// TwinCAT 3 PLC project MasterController
// ProgramVersion: 3.1.4024.0
// libraries:
//   Tc2_EtherCAT, * (Beckhoff Automation GmbH)
//   Tc2_Math, * (Beckhoff Automation GmbH)
//   Tc2_Standard, * (Beckhoff Automation GmbH)
//   Tc2_System, * (Beckhoff Automation GmbH)
//   Tc2_Utilities, * (Beckhoff Automation GmbH)
//   Tc3_Module, * (Beckhoff Automation GmbH)
// project tree:
//   AgiMaths/Frames/ DHTrans.TcPOU (not stored), invFrame.TcPOU, rotX.TcPOU, rotY.TcPOU, rotZ.TcPOU, transform.TcPOU
//   AgiMaths/MatrixLib/ angAxis2Rot.TcPOU, cross.TcPOU (not stored), Det5.TcPOU, Det6.TcPOU, Det7.TcPOU (not stored), invMat6.TcPOU, invMat6Old.TcPOU (not stored), invMat3.TcPOU, invMat7.TcPOU, Mat3T.TcPOU (not stored), matAdd.TcPOU, matMultiNum.TcPOU, matMultiply.TcPOU, matMultiVec.TcPOU, matSelfAdd.TcPOU, matSelfSub.TcPOU, matSub.TcPOU, matTranspose.TcPOU, rot2AngAxis.TcPOU, norm.TcPOU, normalize.TcPOU, vecAdd.TcPOU, vecDot.TcPOU, vecMultiNum.TcPOU, vecSelfAdd.TcPOU, vecSelfMultiNum.TcPOU, vecSelfSub.TcPOU, vecSub.TcPOU
//   AgiMaths/ sign.TcPOU (not stored), addVec7.TcPOU (not stored), atan2.TcPOU, cot.TcPOU (not stored)
//   DUTs/Enum/ E_InstruEnergyCtrlWord.TcDUT, E_InstrumentEnergyType.TcDUT, E_InstrumentType.TcDUT, E_MasterArmState.TcDUT, E_MatchedSlaveArmIdx.TcDUT (not stored), E_SlaveArmState.TcDUT, E_DriverCtrlWord.TcDUT (not stored), E_DriverOPMode.TcDUT, E_DriverStatusWord.TcDUT (not stored)
//   DUTs/Structure/MasterSlaveCommunication/ ST_MasterStatus.TcDUT, ST_SlaveStatus.TcDUT
//   DUTs/Structure/ ST_EtherCATState.TcDUT, ST_InstruStatus.TcDUT, ST_MatchedMasterArmIdx.TcDUT, ST_ArmCtrlCmds.TcDUT (not stored), ST_MasterInputDataPool.TcDUT, ST_Frame.TcDUT (not stored)
//   DUTs/Structure/TasksCommunication/ ST_CartUIData.TcDUT, ST_MasterDynaData.TcDUT, ST_MasterUIData.TcDUT, ST_CartStatus.TcDUT, ST_MasterJointData.TcDUT, ST_MotorInputs.TcDUT (not stored), ST_MotorOutputs.TcDUT, ST_SlaveJointData.TcDUT, ST_SafetyData.TcDUT, ST_CartJointData.TcDUT
//   DUTs/Structure/UICommunication/ ST_arm_distribution.TcDUT, ST_ergonCtrlEnable.TcDUT, ST_ergonomicCtrlData.TcDUT, ST_instrument_info.TcDUT, ST_scope_info.TcDUT
//   DUTs/Type/ Vec7b.TcDUT, Mat34.TcDUT, Mat37.TcDUT, Mat43.TcDUT, Mat4d.TcDUT, Mat5d.TcDUT, Mat67.TcDUT (not stored), Mat6d.TcDUT (not stored), Mat76.TcDUT (not stored), Mat7d.TcDUT (not stored), Vec4d.TcDUT, Vec4i.TcDUT, Vec6i.TcDUT, Vec4b.TcDUT, Vec7di.TcDUT, Vec8d.TcDUT, Mat3d.TcDUT (not stored), Vec3d.TcDUT (not stored), Vec6d.TcDUT (not stored), Vec7d.TcDUT, Vec7i.TcDUT
//   FBs_Auxiliary/ FB_GripAngleCalc.TcPOU, FB_HandClutchCheck.TcPOU, FB_IOCheck.TcPOU, FB_RiseEdgeCheck.TcPOU, FB_IOToggleCheck.TcPOU, FB_MSCtrlTriggerCheck.TcPOU, FB_slaveConnectionCheck.TcPOU, FB_TON.TcPOU
//   FBs_BasicControllers/ FB_boundaryForceFeedback.TcPOU, FB_PID.TcPOU (not stored), FB_RedunJntControl.TcPOU
//   FBs_Observer/ FB_JntObserver.TcPOU
//   FBs_RobotDynamics/ FB_MasterDynamic.TcPOU, FB_MasterFriciton.TcPOU, FB_MasterGravity.TcPOU
//   FBs_Robots/ FB_ArmJoint.TcPOU, FB_CartJoint.TcPOU, FB_JointBase.TcPOU, FB_MasterCart.TcPOU, FB_MasterArm.TcPOU, FB_MasterRobot.TcPOU
//   FBs_StateControllers/ FB_EndoscopeController.TcPOU, FB_StateCtrlClutch.TcPOU, FB_StateCtrlEndoscope.TcPOU, FB_StateCtrlCart.TcPOU, FB_StateCtrlDisable.TcPOU, FB_StateCtrlGraCali.TcPOU, FB_StateCtrlMatching.TcPOU, FB_StateCtrlHome.TcPOU, FB_StateCtrlError.TcPOU, FB_StateCtrlPerformance.TcPOU, FB_StateCtrlReady.TcPOU, FB_StateCtrlMasterSlave.TcPOU, FB_StateCtrlTest.TcPOU, FB_StateCtrlInit.TcPOU, FB_StateCtrlStandBy.TcPOU, FB_MasterArmCtrlBase.TcPOU, I_MasterArmCtrl.TcIO
//   FBs_TrajectoryPlanning/ FB_BasicDoubleS.TcPOU, FB_trajBase.TcPOU, FB_TrajMoveJ.TcPOU, linear_trajectory_with_quintic_polynomial_blends.TcPOU (not stored), quintic_spline_curve.TcPOU (not stored), Quintic_spline_curve_factor.TcPOU (not stored), TrapezoIDal_velocity_trajectory.TcPOU (not stored)
//   FBs_TrajectoryPlanning/OTG/ FB_secOrdTrajFilter.TcPOU, FB_thirdOrdTrajFilter.TcPOU (not stored)
//   FBs_Filters/ FB_LowPassFilter.TcPOU
//   GVLs/Arms/ GVL_ArmDynamics.TcGVL, GVL_ArmJointCaliData.TcGVL, GVL_ArmKinematic.TcGVL, GVL_ControlParameters.TcGVL, GVL_ArmJointParameters.TcGVL
//   GVLs/Cart/ GVL_CartJointCaliData.TcGVL, GVL_CartJointParameters.TcGVL
//   GVLs/Configs/Robot3/ GVL_ArmDynamics_3.TcGVL, GVL_ArmJointCaliData_3.TcGVL, GVL_CartJointCaliData_3.TcGVL
//   GVLs/Configs/Robot4/ GVL_ArmDynamics_4.TcGVL, GVL_ArmJointCaliData_4.TcGVL, GVL_CartJointCaliData_4_1.TcGVL
//   GVLs/Configs/Robot5/ GVL_ArmDynamics_5.TcGVL, GVL_ArmJointCaliData_5.TcGVL, GVL_CartJointCaliData_5.TcGVL
//   GVLs/Configs/Robot6/ GVL_ArmDynamics_6.TcGVL, GVL_ArmJointCaliData_6.TcGVL, GVL_CartJointCaliData_6.TcGVL
//   GVLs/ GVL_interactUI.TcGVL, GVL_MathDefine.TcGVL, GVL_SafetyParameters.TcGVL, GVL_SystemParameters.TcGVL
//   Mains/ CartControl.TcPOU, SafetyCheck.TcPOU, MasterArmControl.TcPOU, RobotDynamics.TcPOU
//   SafetyCheck/ ASSERT.TcPOU, Fb_dataRecord.TcPOU, FB_EtherCATCheck.TcPOU, Fb_SafetyCheck.TcPOU, FB_Writer.TcPOU
//   SafetyCheck/safetyCheckDUT/ checkDelay.TcDUT, checkDelayTime.TcDUT, checkInputVariable.TcDUT, checkPermit.TcDUT, ST_Buffer.TcDUT, T_Buffer.TcDUT
//   Sandbox/ FB_CartCheck.TcPOU, FB_MasterArmCheck.TcPOU, FB_RedunJntControl_bak2.TcPOU, FB_RedunJntControl_bak.TcPOU
//   / TaskArmControl.TcTTO, TaskCartControl.TcTTO, TaskDynamic.TcTTO, TaskSafetyCheck.TcTTO
// real-time tasks:
//   TASK TaskArmControl: cycle T#250us, priority 1, ADS port 350
//   TASK TaskDynamic: cycle T#1ms, priority 2, ADS port 351
//   TASK TaskSafetyCheck: cycle T#1ms, priority 5, ADS port 352
//   TASK TaskCartControl: cycle T#1ms, priority 4, ADS port 353
// I/O:
//   DEVICE RightArm (EtherCAT), AmsNetId 192.168.0.10.9.1
//     Term 19 (EK1100) [EK1100 EtherCAT Coupler (2A E-Bus)]
//       Term 20 (EL6070-0033) [EL6070-0033 1Ch. Licence key terminal, individual licences]
//       Term 21 (EL1008) [EL1008 8Ch. Dig. Input 24V, 3ms]
//       Term 22 (EL1008) [EL1008 8Ch. Dig. Input 24V, 3ms]
//       Term 23 (EL1008) [EL1008 8Ch. Dig. Input 24V, 3ms]
//       Term 24 (EL2008-0015) [EL2008-0015 8K. Dig. Ausgang 24V DC, 0.35A, nicht kurzschlussfest]
//       Term 25 (EK1122) [EK1122 2 port EtherCAT junction]
//         CartArmSet [AX58200_MotorControl_1axis]
//         CartMonitorLift [AX58200_MotorControl_1axis]
//         CartPedal [AX58200_MotorControl_1axis]
//         CartMonitorRotate [AX58200_MotorControl_1axis]
//     Joint1 [AX58200_MotorControl_1axis]
//     Joint2 [AX58200_MotorControl_1axis]
//     Joint3 [AX58200_MotorControl_1axis]
//     Joint4 [AX58200_MotorControl_1axis]
//     Joint5 [AX58200_MotorControl_1axis]
//     Joint6 [AX58200_MotorControl_1axis]
//     Joint7 [AX58200_MotorControl_1axis]
//   DEVICE LeftArm (EtherCAT), AmsNetId 192.168.0.10.4.1
//     Joint1 [AX58200_MotorControl_1axis]
//     Joint2 [AX58200_MotorControl_1axis]
//     Joint3 [AX58200_MotorControl_1axis]
//     Joint4 [AX58200_MotorControl_1axis]
//     Joint5 [AX58200_MotorControl_1axis]
//     Joint6 [AX58200_MotorControl_1axis]
//     Joint7 [AX58200_MotorControl_1axis]
//   DEVICE MSCommunication (EtherCAT), AmsNetId 192.168.0.10.7.1
//     Box 45 (AX58200_MotorControl) [AX58200_MotorControl2021.9.13]
//     Box 46 (EL6695-0002) [EL6695 EtherCAT Bridge terminal (Secondary)]
// variable links:
//   MasterController/MasterController Instance <-> LeftArm (EtherCAT)/Joint1
//     TaskArmControl Inputs/MasterArmControl.m_masterRobot.m_masterArms[1].m_joints[1].m_motorInputs/m_current <-> TxPdoMappingCspCsv/Torque actual value
//     TaskArmControl Inputs/MasterArmControl.m_masterRobot.m_masterArms[1].m_joints[1].m_motorInputs/m_driverError <-> TxPdoMappingCspCsv/digital input
//     TaskArmControl Inputs/MasterArmControl.m_masterRobot.m_masterArms[1].m_joints[1].m_motorInputs/m_linkEncoder <-> TxPdoMappingCspCsv/ENC2
//     TaskArmControl Inputs/MasterArmControl.m_masterRobot.m_masterArms[1].m_joints[1].m_motorInputs/m_motorEncoder <-> TxPdoMappingCspCsv/Position actual value
//     TaskArmControl Inputs/MasterArmControl.m_masterRobot.m_masterArms[1].m_joints[1].m_motorInputs/m_statusWord <-> TxPdoMappingCspCsv/Statusword
//     TaskArmControl Outputs/MasterArmControl.m_masterRobot.m_masterArms[1].m_joints[1].m_motorOutputs/m_cmdCurrent <-> RxPdoMappingCspCsv/Target torque
//     TaskArmControl Outputs/MasterArmControl.m_masterRobot.m_masterArms[1].m_joints[1].m_motorOutputs/m_cmdMotorEncoder <-> RxPdoMappingCspCsv/Target position
//     TaskArmControl Outputs/MasterArmControl.m_masterRobot.m_masterArms[1].m_joints[1].m_motorOutputs/m_controlWord <-> RxPdoMappingCspCsv/Controlword
//     TaskArmControl Outputs/MasterArmControl.m_masterRobot.m_masterArms[1].m_joints[1].m_motorOutputs/m_opMode <-> RxPdoMappingCspCsv/Modes of operation
//   MasterController/MasterController Instance <-> LeftArm (EtherCAT)/Joint2
//     TaskArmControl Inputs/MasterArmControl.m_masterRobot.m_masterArms[1].m_joints[2].m_motorInputs/m_current <-> TxPdoMappingCspCsv/Torque actual value
//     TaskArmControl Inputs/MasterArmControl.m_masterRobot.m_masterArms[1].m_joints[2].m_motorInputs/m_driverError <-> TxPdoMappingCspCsv/digital input
//     TaskArmControl Inputs/MasterArmControl.m_masterRobot.m_masterArms[1].m_joints[2].m_motorInputs/m_linkEncoder <-> TxPdoMappingCspCsv/ENC2
//     TaskArmControl Inputs/MasterArmControl.m_masterRobot.m_masterArms[1].m_joints[2].m_motorInputs/m_motorEncoder <-> TxPdoMappingCspCsv/Position actual value
//     TaskArmControl Inputs/MasterArmControl.m_masterRobot.m_masterArms[1].m_joints[2].m_motorInputs/m_statusWord <-> TxPdoMappingCspCsv/Statusword
//     TaskArmControl Outputs/MasterArmControl.m_masterRobot.m_masterArms[1].m_joints[2].m_motorOutputs/m_cmdCurrent <-> RxPdoMappingCspCsv/Target torque
//     TaskArmControl Outputs/MasterArmControl.m_masterRobot.m_masterArms[1].m_joints[2].m_motorOutputs/m_cmdMotorEncoder <-> RxPdoMappingCspCsv/Target position
//     TaskArmControl Outputs/MasterArmControl.m_masterRobot.m_masterArms[1].m_joints[2].m_motorOutputs/m_controlWord <-> RxPdoMappingCspCsv/Controlword
//     TaskArmControl Outputs/MasterArmControl.m_masterRobot.m_masterArms[1].m_joints[2].m_motorOutputs/m_opMode <-> RxPdoMappingCspCsv/Modes of operation
//   MasterController/MasterController Instance <-> LeftArm (EtherCAT)/Joint3
//     TaskArmControl Inputs/MasterArmControl.m_masterRobot.m_masterArms[1].m_joints[3].m_motorInputs/m_current <-> TxPdoMappingCspCsv/Torque actual value
//     TaskArmControl Inputs/MasterArmControl.m_masterRobot.m_masterArms[1].m_joints[3].m_motorInputs/m_driverError <-> TxPdoMappingCspCsv/digital input
//     TaskArmControl Inputs/MasterArmControl.m_masterRobot.m_masterArms[1].m_joints[3].m_motorInputs/m_linkEncoder <-> TxPdoMappingCspCsv/ENC2
//     TaskArmControl Inputs/MasterArmControl.m_masterRobot.m_masterArms[1].m_joints[3].m_motorInputs/m_motorEncoder <-> TxPdoMappingCspCsv/Position actual value
//     TaskArmControl Inputs/MasterArmControl.m_masterRobot.m_masterArms[1].m_joints[3].m_motorInputs/m_statusWord <-> TxPdoMappingCspCsv/Statusword
//     TaskArmControl Outputs/MasterArmControl.m_masterRobot.m_masterArms[1].m_joints[3].m_motorOutputs/m_cmdCurrent <-> RxPdoMappingCspCsv/Target torque
//     TaskArmControl Outputs/MasterArmControl.m_masterRobot.m_masterArms[1].m_joints[3].m_motorOutputs/m_cmdMotorEncoder <-> RxPdoMappingCspCsv/Target position
//     TaskArmControl Outputs/MasterArmControl.m_masterRobot.m_masterArms[1].m_joints[3].m_motorOutputs/m_controlWord <-> RxPdoMappingCspCsv/Controlword
//     TaskArmControl Outputs/MasterArmControl.m_masterRobot.m_masterArms[1].m_joints[3].m_motorOutputs/m_opMode <-> RxPdoMappingCspCsv/Modes of operation
//   MasterController/MasterController Instance <-> LeftArm (EtherCAT)/Joint4
//     TaskArmControl Inputs/MasterArmControl.m_masterRobot.m_masterArms[1].m_joints[4].m_motorInputs/m_current <-> TxPdoMappingCspCsv/Torque actual value
//     TaskArmControl Inputs/MasterArmControl.m_masterRobot.m_masterArms[1].m_joints[4].m_motorInputs/m_driverError <-> TxPdoMappingCspCsv/digital input
//     TaskArmControl Inputs/MasterArmControl.m_masterRobot.m_masterArms[1].m_joints[4].m_motorInputs/m_motorEncoder <-> TxPdoMappingCspCsv/Position actual value
//     TaskArmControl Inputs/MasterArmControl.m_masterRobot.m_masterArms[1].m_joints[4].m_motorInputs/m_statusWord <-> TxPdoMappingCspCsv/Statusword
//     TaskArmControl Outputs/MasterArmControl.m_masterRobot.m_masterArms[1].m_joints[4].m_motorOutputs/m_cmdCurrent <-> RxPdoMappingCspCsv/Target torque
//     TaskArmControl Outputs/MasterArmControl.m_masterRobot.m_masterArms[1].m_joints[4].m_motorOutputs/m_cmdMotorEncoder <-> RxPdoMappingCspCsv/Target position
//     TaskArmControl Outputs/MasterArmControl.m_masterRobot.m_masterArms[1].m_joints[4].m_motorOutputs/m_controlWord <-> RxPdoMappingCspCsv/Controlword
//     TaskArmControl Outputs/MasterArmControl.m_masterRobot.m_masterArms[1].m_joints[4].m_motorOutputs/m_opMode <-> RxPdoMappingCspCsv/Modes of operation
//   MasterController/MasterController Instance <-> LeftArm (EtherCAT)/Joint5
//     TaskArmControl Inputs/MasterArmControl.m_masterRobot.m_masterArms[1].m_joints[4].m_motorInputs/m_linkEncoder <-> TxPdoMappingCspCsv/Velocity actual value
//     TaskArmControl Inputs/MasterArmControl.m_masterRobot.m_masterArms[1].m_joints[5].m_motorInputs/m_current <-> TxPdoMappingCspCsv/Torque actual value
//     TaskArmControl Inputs/MasterArmControl.m_masterRobot.m_masterArms[1].m_joints[5].m_motorInputs/m_driverError <-> TxPdoMappingCspCsv/digital input
//     TaskArmControl Inputs/MasterArmControl.m_masterRobot.m_masterArms[1].m_joints[5].m_motorInputs/m_linkEncoder <-> TxPdoMappingCspCsv/ENC2
//     TaskArmControl Inputs/MasterArmControl.m_masterRobot.m_masterArms[1].m_joints[5].m_motorInputs/m_motorEncoder <-> TxPdoMappingCspCsv/Position actual value
//     TaskArmControl Inputs/MasterArmControl.m_masterRobot.m_masterArms[1].m_joints[5].m_motorInputs/m_statusWord <-> TxPdoMappingCspCsv/Statusword
//     TaskArmControl Outputs/MasterArmControl.m_masterRobot.m_masterArms[1].m_joints[5].m_motorOutputs/m_cmdCurrent <-> RxPdoMappingCspCsv/Target torque
//     TaskArmControl Outputs/MasterArmControl.m_masterRobot.m_masterArms[1].m_joints[5].m_motorOutputs/m_cmdMotorEncoder <-> RxPdoMappingCspCsv/Target position
//     TaskArmControl Outputs/MasterArmControl.m_masterRobot.m_masterArms[1].m_joints[5].m_motorOutputs/m_controlWord <-> RxPdoMappingCspCsv/Controlword
//     TaskArmControl Outputs/MasterArmControl.m_masterRobot.m_masterArms[1].m_joints[5].m_motorOutputs/m_opMode <-> RxPdoMappingCspCsv/Modes of operation
//   MasterController/MasterController Instance <-> LeftArm (EtherCAT)/Joint6
//     TaskArmControl Inputs/MasterArmControl.m_masterRobot.m_masterArms[1].m_joints[6].m_motorInputs/m_current <-> TxPdoMappingCspCsv/Torque actual value
//     TaskArmControl Inputs/MasterArmControl.m_masterRobot.m_masterArms[1].m_joints[6].m_motorInputs/m_driverError <-> TxPdoMappingCspCsv/digital input
//     TaskArmControl Inputs/MasterArmControl.m_masterRobot.m_masterArms[1].m_joints[6].m_motorInputs/m_linkEncoder <-> TxPdoMappingCspCsv/ENC2
//     TaskArmControl Inputs/MasterArmControl.m_masterRobot.m_masterArms[1].m_joints[6].m_motorInputs/m_motorEncoder <-> TxPdoMappingCspCsv/Position actual value
//     TaskArmControl Inputs/MasterArmControl.m_masterRobot.m_masterArms[1].m_joints[6].m_motorInputs/m_statusWord <-> TxPdoMappingCspCsv/Statusword
//     TaskArmControl Outputs/MasterArmControl.m_masterRobot.m_masterArms[1].m_joints[6].m_motorOutputs/m_cmdCurrent <-> RxPdoMappingCspCsv/Target torque
//     TaskArmControl Outputs/MasterArmControl.m_masterRobot.m_masterArms[1].m_joints[6].m_motorOutputs/m_cmdMotorEncoder <-> RxPdoMappingCspCsv/Target position
//     TaskArmControl Outputs/MasterArmControl.m_masterRobot.m_masterArms[1].m_joints[6].m_motorOutputs/m_controlWord <-> RxPdoMappingCspCsv/Controlword
//     TaskArmControl Outputs/MasterArmControl.m_masterRobot.m_masterArms[1].m_joints[6].m_motorOutputs/m_opMode <-> RxPdoMappingCspCsv/Modes of operation
//   MasterController/MasterController Instance <-> LeftArm (EtherCAT)/Joint7
//     TaskArmControl Inputs/MasterArmControl.m_masterRobot.m_masterArms[1].m_gripHallSensorIO <-> TxPdoMappingCspCsv/analog input
//     TaskArmControl Inputs/MasterArmControl.m_masterRobot.m_masterArms[1].m_handClutchIO <-> TxPdoMappingCspCsv/digital input
//     TaskArmControl Inputs/MasterArmControl.m_masterRobot.m_masterArms[1].m_joints[7].m_motorInputs/m_current <-> TxPdoMappingCspCsv/Torque actual value
//     TaskArmControl Inputs/MasterArmControl.m_masterRobot.m_masterArms[1].m_joints[7].m_motorInputs/m_linkEncoder <-> TxPdoMappingCspCsv/ENC2
//     TaskArmControl Inputs/MasterArmControl.m_masterRobot.m_masterArms[1].m_joints[7].m_motorInputs/m_motorEncoder <-> TxPdoMappingCspCsv/Position actual value
//     TaskArmControl Inputs/MasterArmControl.m_masterRobot.m_masterArms[1].m_joints[7].m_motorInputs/m_statusWord <-> TxPdoMappingCspCsv/Statusword
//     TaskArmControl Outputs/MasterArmControl.m_masterRobot.m_masterArms[1].m_joints[7].m_motorOutputs/m_cmdCurrent <-> RxPdoMappingCspCsv/Target torque
//     TaskArmControl Outputs/MasterArmControl.m_masterRobot.m_masterArms[1].m_joints[7].m_motorOutputs/m_cmdMotorEncoder <-> RxPdoMappingCspCsv/Target position
//     TaskArmControl Outputs/MasterArmControl.m_masterRobot.m_masterArms[1].m_joints[7].m_motorOutputs/m_controlWord <-> RxPdoMappingCspCsv/Controlword
//     TaskArmControl Outputs/MasterArmControl.m_masterRobot.m_masterArms[1].m_joints[7].m_motorOutputs/m_opMode <-> RxPdoMappingCspCsv/Modes of operation
//   MasterController/MasterController Instance <-> MSCommunication (EtherCAT)/Box 45 (AX58200_MotorControl)
//     TaskCartControl Outputs/CartControl.m_masterCart.m_elecKnifeCtrlWord <-> RxPdoMappingCspCsv/Target velocity
//   MasterController/MasterController Instance <-> MSCommunication (EtherCAT)/Box 46 (EL6695-0002)
//     TaskArmControl Inputs/MasterArmControl.m_slaveRobotData <-> IO Inputs/SlaveRobotData
//     TaskArmControl Outputs/MasterArmControl.m_masterRobotData <-> IO Outputs/MasterRobotData
//   MasterController/MasterController Instance <-> RightArm (EtherCAT)/Joint1
//     TaskArmControl Inputs/MasterArmControl.m_masterRobot.m_masterArms[2].m_joints[1].m_motorInputs/m_current <-> TxPdoMappingCspCsv/Torque actual value
//     TaskArmControl Inputs/MasterArmControl.m_masterRobot.m_masterArms[2].m_joints[1].m_motorInputs/m_driverError <-> TxPdoMappingCspCsv/digital input
//     TaskArmControl Inputs/MasterArmControl.m_masterRobot.m_masterArms[2].m_joints[1].m_motorInputs/m_linkEncoder <-> TxPdoMappingCspCsv/ENC2
//     TaskArmControl Inputs/MasterArmControl.m_masterRobot.m_masterArms[2].m_joints[1].m_motorInputs/m_motorEncoder <-> TxPdoMappingCspCsv/Position actual value
//     TaskArmControl Inputs/MasterArmControl.m_masterRobot.m_masterArms[2].m_joints[1].m_motorInputs/m_statusWord <-> TxPdoMappingCspCsv/Statusword
//     TaskArmControl Outputs/MasterArmControl.m_masterRobot.m_masterArms[2].m_joints[1].m_motorOutputs/m_cmdCurrent <-> RxPdoMappingCspCsv/Target torque
//     TaskArmControl Outputs/MasterArmControl.m_masterRobot.m_masterArms[2].m_joints[1].m_motorOutputs/m_cmdMotorEncoder <-> RxPdoMappingCspCsv/Target position
//     TaskArmControl Outputs/MasterArmControl.m_masterRobot.m_masterArms[2].m_joints[1].m_motorOutputs/m_controlWord <-> RxPdoMappingCspCsv/Controlword
//     TaskArmControl Outputs/MasterArmControl.m_masterRobot.m_masterArms[2].m_joints[1].m_motorOutputs/m_opMode <-> RxPdoMappingCspCsv/Modes of operation
//   MasterController/MasterController Instance <-> RightArm (EtherCAT)/Joint2
//     TaskArmControl Inputs/MasterArmControl.m_masterRobot.m_masterArms[2].m_joints[2].m_motorInputs/m_current <-> TxPdoMappingCspCsv/Torque actual value
//     TaskArmControl Inputs/MasterArmControl.m_masterRobot.m_masterArms[2].m_joints[2].m_motorInputs/m_driverError <-> TxPdoMappingCspCsv/digital input
//     TaskArmControl Inputs/MasterArmControl.m_masterRobot.m_masterArms[2].m_joints[2].m_motorInputs/m_linkEncoder <-> TxPdoMappingCspCsv/ENC2
//     TaskArmControl Inputs/MasterArmControl.m_masterRobot.m_masterArms[2].m_joints[2].m_motorInputs/m_motorEncoder <-> TxPdoMappingCspCsv/Position actual value
//     TaskArmControl Inputs/MasterArmControl.m_masterRobot.m_masterArms[2].m_joints[2].m_motorInputs/m_statusWord <-> TxPdoMappingCspCsv/Statusword
//     TaskArmControl Outputs/MasterArmControl.m_masterRobot.m_masterArms[2].m_joints[2].m_motorOutputs/m_cmdCurrent <-> RxPdoMappingCspCsv/Target torque
//     TaskArmControl Outputs/MasterArmControl.m_masterRobot.m_masterArms[2].m_joints[2].m_motorOutputs/m_cmdMotorEncoder <-> RxPdoMappingCspCsv/Target position
//     TaskArmControl Outputs/MasterArmControl.m_masterRobot.m_masterArms[2].m_joints[2].m_motorOutputs/m_controlWord <-> RxPdoMappingCspCsv/Controlword
//     TaskArmControl Outputs/MasterArmControl.m_masterRobot.m_masterArms[2].m_joints[2].m_motorOutputs/m_opMode <-> RxPdoMappingCspCsv/Modes of operation
//   MasterController/MasterController Instance <-> RightArm (EtherCAT)/Joint3
//     TaskArmControl Inputs/MasterArmControl.m_masterRobot.m_masterArms[2].m_joints[3].m_motorInputs/m_current <-> TxPdoMappingCspCsv/Torque actual value
//     TaskArmControl Inputs/MasterArmControl.m_masterRobot.m_masterArms[2].m_joints[3].m_motorInputs/m_driverError <-> TxPdoMappingCspCsv/digital input
//     TaskArmControl Inputs/MasterArmControl.m_masterRobot.m_masterArms[2].m_joints[3].m_motorInputs/m_linkEncoder <-> TxPdoMappingCspCsv/ENC2
//     TaskArmControl Inputs/MasterArmControl.m_masterRobot.m_masterArms[2].m_joints[3].m_motorInputs/m_motorEncoder <-> TxPdoMappingCspCsv/Position actual value
//     TaskArmControl Inputs/MasterArmControl.m_masterRobot.m_masterArms[2].m_joints[3].m_motorInputs/m_statusWord <-> TxPdoMappingCspCsv/Statusword
//     TaskArmControl Outputs/MasterArmControl.m_masterRobot.m_masterArms[2].m_joints[3].m_motorOutputs/m_cmdCurrent <-> RxPdoMappingCspCsv/Target torque
//     TaskArmControl Outputs/MasterArmControl.m_masterRobot.m_masterArms[2].m_joints[3].m_motorOutputs/m_cmdMotorEncoder <-> RxPdoMappingCspCsv/Target position
//     TaskArmControl Outputs/MasterArmControl.m_masterRobot.m_masterArms[2].m_joints[3].m_motorOutputs/m_controlWord <-> RxPdoMappingCspCsv/Controlword
//     TaskArmControl Outputs/MasterArmControl.m_masterRobot.m_masterArms[2].m_joints[3].m_motorOutputs/m_opMode <-> RxPdoMappingCspCsv/Modes of operation
//   MasterController/MasterController Instance <-> RightArm (EtherCAT)/Joint4
//     TaskArmControl Inputs/MasterArmControl.m_masterRobot.m_masterArms[2].m_joints[4].m_motorInputs/m_current <-> TxPdoMappingCspCsv/Torque actual value
//     TaskArmControl Inputs/MasterArmControl.m_masterRobot.m_masterArms[2].m_joints[4].m_motorInputs/m_driverError <-> TxPdoMappingCspCsv/digital input
//     TaskArmControl Inputs/MasterArmControl.m_masterRobot.m_masterArms[2].m_joints[4].m_motorInputs/m_motorEncoder <-> TxPdoMappingCspCsv/Position actual value
//     TaskArmControl Inputs/MasterArmControl.m_masterRobot.m_masterArms[2].m_joints[4].m_motorInputs/m_statusWord <-> TxPdoMappingCspCsv/Statusword
//     TaskArmControl Outputs/MasterArmControl.m_masterRobot.m_masterArms[2].m_joints[4].m_motorOutputs/m_cmdCurrent <-> RxPdoMappingCspCsv/Target torque
//     TaskArmControl Outputs/MasterArmControl.m_masterRobot.m_masterArms[2].m_joints[4].m_motorOutputs/m_cmdMotorEncoder <-> RxPdoMappingCspCsv/Target position
//     TaskArmControl Outputs/MasterArmControl.m_masterRobot.m_masterArms[2].m_joints[4].m_motorOutputs/m_controlWord <-> RxPdoMappingCspCsv/Controlword
//     TaskArmControl Outputs/MasterArmControl.m_masterRobot.m_masterArms[2].m_joints[4].m_motorOutputs/m_opMode <-> RxPdoMappingCspCsv/Modes of operation
//   MasterController/MasterController Instance <-> RightArm (EtherCAT)/Joint5
//     TaskArmControl Inputs/MasterArmControl.m_masterRobot.m_masterArms[2].m_joints[4].m_motorInputs/m_linkEncoder <-> TxPdoMappingCspCsv/Velocity actual value
//     TaskArmControl Inputs/MasterArmControl.m_masterRobot.m_masterArms[2].m_joints[5].m_motorInputs/m_current <-> TxPdoMappingCspCsv/Torque actual value
//     TaskArmControl Inputs/MasterArmControl.m_masterRobot.m_masterArms[2].m_joints[5].m_motorInputs/m_driverError <-> TxPdoMappingCspCsv/digital input
//     TaskArmControl Inputs/MasterArmControl.m_masterRobot.m_masterArms[2].m_joints[5].m_motorInputs/m_linkEncoder <-> TxPdoMappingCspCsv/ENC2
//     TaskArmControl Inputs/MasterArmControl.m_masterRobot.m_masterArms[2].m_joints[5].m_motorInputs/m_motorEncoder <-> TxPdoMappingCspCsv/Position actual value
//     TaskArmControl Inputs/MasterArmControl.m_masterRobot.m_masterArms[2].m_joints[5].m_motorInputs/m_statusWord <-> TxPdoMappingCspCsv/Statusword
//     TaskArmControl Outputs/MasterArmControl.m_masterRobot.m_masterArms[2].m_joints[5].m_motorOutputs/m_cmdCurrent <-> RxPdoMappingCspCsv/Target torque
//     TaskArmControl Outputs/MasterArmControl.m_masterRobot.m_masterArms[2].m_joints[5].m_motorOutputs/m_cmdMotorEncoder <-> RxPdoMappingCspCsv/Target position
//     TaskArmControl Outputs/MasterArmControl.m_masterRobot.m_masterArms[2].m_joints[5].m_motorOutputs/m_controlWord <-> RxPdoMappingCspCsv/Controlword
//     TaskArmControl Outputs/MasterArmControl.m_masterRobot.m_masterArms[2].m_joints[5].m_motorOutputs/m_opMode <-> RxPdoMappingCspCsv/Modes of operation
//   MasterController/MasterController Instance <-> RightArm (EtherCAT)/Joint6
//     TaskArmControl Inputs/MasterArmControl.m_masterRobot.m_masterArms[2].m_joints[6].m_motorInputs/m_current <-> TxPdoMappingCspCsv/Torque actual value
//     TaskArmControl Inputs/MasterArmControl.m_masterRobot.m_masterArms[2].m_joints[6].m_motorInputs/m_driverError <-> TxPdoMappingCspCsv/digital input
//     TaskArmControl Inputs/MasterArmControl.m_masterRobot.m_masterArms[2].m_joints[6].m_motorInputs/m_linkEncoder <-> TxPdoMappingCspCsv/ENC2
//     TaskArmControl Inputs/MasterArmControl.m_masterRobot.m_masterArms[2].m_joints[6].m_motorInputs/m_motorEncoder <-> TxPdoMappingCspCsv/Position actual value
//     TaskArmControl Inputs/MasterArmControl.m_masterRobot.m_masterArms[2].m_joints[6].m_motorInputs/m_statusWord <-> TxPdoMappingCspCsv/Statusword
//     TaskArmControl Outputs/MasterArmControl.m_masterRobot.m_masterArms[2].m_joints[6].m_motorOutputs/m_cmdCurrent <-> RxPdoMappingCspCsv/Target torque
//     TaskArmControl Outputs/MasterArmControl.m_masterRobot.m_masterArms[2].m_joints[6].m_motorOutputs/m_cmdMotorEncoder <-> RxPdoMappingCspCsv/Target position
//     TaskArmControl Outputs/MasterArmControl.m_masterRobot.m_masterArms[2].m_joints[6].m_motorOutputs/m_controlWord <-> RxPdoMappingCspCsv/Controlword
//     TaskArmControl Outputs/MasterArmControl.m_masterRobot.m_masterArms[2].m_joints[6].m_motorOutputs/m_opMode <-> RxPdoMappingCspCsv/Modes of operation
//   MasterController/MasterController Instance <-> RightArm (EtherCAT)/Joint7
//     TaskArmControl Inputs/MasterArmControl.m_masterRobot.m_masterArms[2].m_gripHallSensorIO <-> TxPdoMappingCspCsv/analog input
//     TaskArmControl Inputs/MasterArmControl.m_masterRobot.m_masterArms[2].m_handClutchIO <-> TxPdoMappingCspCsv/digital input
//     TaskArmControl Inputs/MasterArmControl.m_masterRobot.m_masterArms[2].m_joints[7].m_motorInputs/m_current <-> TxPdoMappingCspCsv/Torque actual value
//     TaskArmControl Inputs/MasterArmControl.m_masterRobot.m_masterArms[2].m_joints[7].m_motorInputs/m_linkEncoder <-> TxPdoMappingCspCsv/ENC2
//     TaskArmControl Inputs/MasterArmControl.m_masterRobot.m_masterArms[2].m_joints[7].m_motorInputs/m_motorEncoder <-> TxPdoMappingCspCsv/Position actual value
//     TaskArmControl Inputs/MasterArmControl.m_masterRobot.m_masterArms[2].m_joints[7].m_motorInputs/m_statusWord <-> TxPdoMappingCspCsv/Statusword
//     TaskArmControl Outputs/MasterArmControl.m_masterRobot.m_masterArms[2].m_joints[7].m_motorOutputs/m_cmdCurrent <-> RxPdoMappingCspCsv/Target torque
//     TaskArmControl Outputs/MasterArmControl.m_masterRobot.m_masterArms[2].m_joints[7].m_motorOutputs/m_cmdMotorEncoder <-> RxPdoMappingCspCsv/Target position
//     TaskArmControl Outputs/MasterArmControl.m_masterRobot.m_masterArms[2].m_joints[7].m_motorOutputs/m_controlWord <-> RxPdoMappingCspCsv/Controlword
//     TaskArmControl Outputs/MasterArmControl.m_masterRobot.m_masterArms[2].m_joints[7].m_motorOutputs/m_opMode <-> RxPdoMappingCspCsv/Modes of operation
//   MasterController/MasterController Instance <-> RightArm (EtherCAT)/Term 19 (EK1100)/Term 21 (EL1008)
//     TaskArmControl Inputs/SafetyCheck.m_stopButton <-> Channel 1/CartControl.m_masterCart.m_stopButton
//     TaskCartControl Inputs/CartControl.m_masterCart.m_armSwitchIO <-> Channel 4/armSwitchIO
//     TaskCartControl Inputs/CartControl.m_masterCart.m_clutchPedalIO <-> Channel 2/CartControl.m_masterCart.m_clutchPedalIO
//     TaskCartControl Inputs/CartControl.m_masterCart.m_electricCoagulLeft <-> Channel 7/Input
//     TaskCartControl Inputs/CartControl.m_masterCart.m_electricCoagulRight <-> Channel 8/Input
//     TaskCartControl Inputs/CartControl.m_masterCart.m_electricCutLeft <-> Channel 5/Input
//     TaskCartControl Inputs/CartControl.m_masterCart.m_electricCutRight <-> Channel 6/Input
//     TaskCartControl Inputs/CartControl.m_masterCart.m_endoScopePedalIO <-> Channel 3/endoscopePedaoIO
//   MasterController/MasterController Instance <-> RightArm (EtherCAT)/Term 19 (EK1100)/Term 22 (EL1008)
//     TaskCartControl Inputs/CartControl.m_masterCart.m_electricCoagulLeftAllow <-> Channel 2/Input
//     TaskCartControl Inputs/CartControl.m_masterCart.m_electricCoagulRightAllow <-> Channel 4/Input
//     TaskCartControl Inputs/CartControl.m_masterCart.m_electricCutLeftAllow <-> Channel 1/Input
//     TaskCartControl Inputs/CartControl.m_masterCart.m_electricCutRightAllow <-> Channel 3/Input
//     TaskCartControl Inputs/CartControl.m_masterCart.m_surgonHeadInIO <-> Channel 5/HeadInIO
//     TaskSafetyCheck Inputs/SafetyCheck.m_cartLockSignalLeft <-> Channel 7/Input
//     TaskSafetyCheck Inputs/SafetyCheck.m_cartLockSignalRight <-> Channel 8/Input
//   MasterController/MasterController Instance <-> RightArm (EtherCAT)/Term 19 (EK1100)/Term 23 (EL1008)
//     TaskCartControl Inputs/CartControl.m_masterCart.m_cartJointCtrlIO[1] <-> Channel 1/monitorUp
//     TaskCartControl Inputs/CartControl.m_masterCart.m_cartJointCtrlIO[2] <-> Channel 2/monitorDown
//     TaskCartControl Inputs/CartControl.m_masterCart.m_cartJointCtrlIO[3] <-> Channel 7/monitorCW
//     TaskCartControl Inputs/CartControl.m_masterCart.m_cartJointCtrlIO[4] <-> Channel 8/monitorCCW
//     TaskCartControl Inputs/CartControl.m_masterCart.m_cartJointCtrlIO[5] <-> Channel 3/armSetUp
//     TaskCartControl Inputs/CartControl.m_masterCart.m_cartJointCtrlIO[6] <-> Channel 4/armSetDown
//     TaskCartControl Inputs/CartControl.m_masterCart.m_cartJointCtrlIO[7] <-> Channel 5/pedalIn
//     TaskCartControl Inputs/CartControl.m_masterCart.m_cartJointCtrlIO[8] <-> Channel 6/pedalOut
//   MasterController/MasterController Instance <-> RightArm (EtherCAT)/Term 19 (EK1100)/Term 25 (EK1122)/CartArmSet
//     TaskCartControl Inputs/CartControl.m_masterCart.m_cartJoints[3].m_motorInputs/m_current <-> TxPdoMappingCspCsv/Torque actual value
//     TaskCartControl Inputs/CartControl.m_masterCart.m_cartJoints[3].m_motorInputs/m_linkEncoder <-> TxPdoMappingCspCsv/ENC2
//     TaskCartControl Inputs/CartControl.m_masterCart.m_cartJoints[3].m_motorInputs/m_motorEncoder <-> TxPdoMappingCspCsv/Position actual value
//     TaskCartControl Inputs/CartControl.m_masterCart.m_cartJoints[3].m_motorInputs/m_statusWord <-> TxPdoMappingCspCsv/Statusword
//     TaskCartControl Outputs/CartControl.m_masterCart.m_cartJoints[3].m_motorOutputs/m_cmdCurrent <-> RxPdoMappingCspCsv/Target torque
//     TaskCartControl Outputs/CartControl.m_masterCart.m_cartJoints[3].m_motorOutputs/m_cmdMotorEncoder <-> RxPdoMappingCspCsv/Target position
//     TaskCartControl Outputs/CartControl.m_masterCart.m_cartJoints[3].m_motorOutputs/m_controlWord <-> RxPdoMappingCspCsv/Controlword
//     TaskCartControl Outputs/CartControl.m_masterCart.m_cartJoints[3].m_motorOutputs/m_opMode <-> RxPdoMappingCspCsv/Modes of operation
//   MasterController/MasterController Instance <-> RightArm (EtherCAT)/Term 19 (EK1100)/Term 25 (EK1122)/CartMonitorLift
//     TaskCartControl Inputs/CartControl.m_masterCart.m_cartJoints[1].m_motorInputs/m_current <-> TxPdoMappingCspCsv/Torque actual value
//     TaskCartControl Inputs/CartControl.m_masterCart.m_cartJoints[1].m_motorInputs/m_linkEncoder <-> TxPdoMappingCspCsv/ENC2
//     TaskCartControl Inputs/CartControl.m_masterCart.m_cartJoints[1].m_motorInputs/m_motorEncoder <-> TxPdoMappingCspCsv/Position actual value
//     TaskCartControl Inputs/CartControl.m_masterCart.m_cartJoints[1].m_motorInputs/m_statusWord <-> TxPdoMappingCspCsv/Statusword
//     TaskCartControl Outputs/CartControl.m_masterCart.m_cartJoints[1].m_motorOutputs/m_cmdCurrent <-> RxPdoMappingCspCsv/Target torque
//     TaskCartControl Outputs/CartControl.m_masterCart.m_cartJoints[1].m_motorOutputs/m_cmdMotorEncoder <-> RxPdoMappingCspCsv/Target position
//     TaskCartControl Outputs/CartControl.m_masterCart.m_cartJoints[1].m_motorOutputs/m_controlWord <-> RxPdoMappingCspCsv/Controlword
//     TaskCartControl Outputs/CartControl.m_masterCart.m_cartJoints[1].m_motorOutputs/m_opMode <-> RxPdoMappingCspCsv/Modes of operation
//   MasterController/MasterController Instance <-> RightArm (EtherCAT)/Term 19 (EK1100)/Term 25 (EK1122)/CartMonitorRotate
//     TaskCartControl Inputs/CartControl.m_masterCart.m_cartJoints[2].m_motorInputs/m_current <-> TxPdoMappingCspCsv/Torque actual value
//     TaskCartControl Inputs/CartControl.m_masterCart.m_cartJoints[2].m_motorInputs/m_linkEncoder <-> TxPdoMappingCspCsv/ENC2
//     TaskCartControl Inputs/CartControl.m_masterCart.m_cartJoints[2].m_motorInputs/m_motorEncoder <-> TxPdoMappingCspCsv/Position actual value
//     TaskCartControl Inputs/CartControl.m_masterCart.m_cartJoints[2].m_motorInputs/m_statusWord <-> TxPdoMappingCspCsv/Statusword
//     TaskCartControl Outputs/CartControl.m_masterCart.m_cartJoints[2].m_motorOutputs/m_cmdCurrent <-> RxPdoMappingCspCsv/Target torque
//     TaskCartControl Outputs/CartControl.m_masterCart.m_cartJoints[2].m_motorOutputs/m_cmdMotorEncoder <-> RxPdoMappingCspCsv/Target position
//     TaskCartControl Outputs/CartControl.m_masterCart.m_cartJoints[2].m_motorOutputs/m_controlWord <-> RxPdoMappingCspCsv/Controlword
//     TaskCartControl Outputs/CartControl.m_masterCart.m_cartJoints[2].m_motorOutputs/m_opMode <-> RxPdoMappingCspCsv/Modes of operation
//   MasterController/MasterController Instance <-> RightArm (EtherCAT)/Term 19 (EK1100)/Term 25 (EK1122)/CartPedal
//     TaskCartControl Inputs/CartControl.m_masterCart.m_cartJoints[4].m_motorInputs/m_current <-> TxPdoMappingCspCsv/Torque actual value
//     TaskCartControl Inputs/CartControl.m_masterCart.m_cartJoints[4].m_motorInputs/m_linkEncoder <-> TxPdoMappingCspCsv/ENC2
//     TaskCartControl Inputs/CartControl.m_masterCart.m_cartJoints[4].m_motorInputs/m_motorEncoder <-> TxPdoMappingCspCsv/Position actual value
//     TaskCartControl Inputs/CartControl.m_masterCart.m_cartJoints[4].m_motorInputs/m_statusWord <-> TxPdoMappingCspCsv/Statusword
//     TaskCartControl Outputs/CartControl.m_masterCart.m_cartJoints[4].m_motorOutputs/m_cmdCurrent <-> RxPdoMappingCspCsv/Target torque
//     TaskCartControl Outputs/CartControl.m_masterCart.m_cartJoints[4].m_motorOutputs/m_cmdMotorEncoder <-> RxPdoMappingCspCsv/Target position
//     TaskCartControl Outputs/CartControl.m_masterCart.m_cartJoints[4].m_motorOutputs/m_controlWord <-> RxPdoMappingCspCsv/Controlword
//     TaskCartControl Outputs/CartControl.m_masterCart.m_cartJoints[4].m_motorOutputs/m_opMode <-> RxPdoMappingCspCsv/Modes of operation
//   MasterController/MasterController Instance <-> MasterController/MasterController Instance
//     TaskArmControl Inputs/MasterArmControl.m_masterInputDataPool.m_cartStatus <-> TaskCartControl Outputs/CartControl.m_cartStatus
//     TaskArmControl Inputs/MasterArmControl.m_masterInputDataPool.m_masterDynaData <-> TaskDynamic Outputs/RobotDynamics.m_masterDynaData
//     TaskArmControl Inputs/MasterArmControl.m_masterInputDataPool.m_safetyData <-> TaskCartControl Outputs/SafetyCheck.m_safetyCheckData
//     TaskDynamic Inputs/RobotDynamics.m_masterJointsData <-> TaskArmControl Outputs/MasterArmControl.m_masterJointsData
//     TaskSafetyCheck Inputs/SafetyCheck.m_cartJointData <-> TaskCartControl Outputs/CartControl.m_cartJointData
//     TaskSafetyCheck Inputs/SafetyCheck.m_cartStatus <-> TaskCartControl Outputs/CartControl.m_cartStatus
//     TaskSafetyCheck Inputs/SafetyCheck.m_masterJointData <-> TaskArmControl Outputs/MasterArmControl.m_masterJointsData
//     TaskSafetyCheck Inputs/SafetyCheck.m_masterStatus <-> TaskArmControl Outputs/MasterArmControl.m_masterStatus

CONFIGURATION MasterController
    RESOURCE PLC ON TwinCAT3
        TASK TaskArmControl(INTERVAL := T#250us, PRIORITY := 1);
        TASK TaskCartControl(INTERVAL := T#1ms, PRIORITY := 4);
        TASK TaskDynamic(INTERVAL := T#1ms, PRIORITY := 2);
        TASK TaskSafetyCheck(INTERVAL := T#1ms, PRIORITY := 5);
        PROGRAM MasterArmControl WITH TaskArmControl : MasterArmControl;
        PROGRAM CartControl WITH TaskCartControl : CartControl;
        PROGRAM RobotDynamics WITH TaskDynamic : RobotDynamics;
        PROGRAM SafetyCheck WITH TaskSafetyCheck : SafetyCheck;
    END_RESOURCE
END_CONFIGURATION

// ---- DUTs/Enum/E_InstruEnergyCtrlWord.TcDUT
TYPE E_InstruEnergyCtrlWord :
(
	EnergyCtrlWord_NoOutput := 0,
	EnergyCtrlWord_isMonopoleCut := 2,
	EnergyCtrlWord_isMonopoleCoagul := 4,
	EnergyCtrlWord_isBipolarCoagul := 1,
	EnergyCtrlWord_isUltraMax := 64,
	EnergyCtrlWord_isUltraMin := 16
);
END_TYPE

// ---- DUTs/Enum/E_InstrumentEnergyType.TcDUT
TYPE E_InstrumentEnergyType :
(
	InstruType_isNull := 0,
	InstruType_isMonopole := 1,
	InstruType_isBipolar := 2,
	InstruType_isUltraKnife := 3
);
END_TYPE

// ---- DUTs/Enum/E_InstrumentType.TcDUT
TYPE E_InstrumentType :
(
	InstruType_UNKNOWM := 0,
	InstruType_CadiereForceps :=7,
	InstruType_NeedleDriver :=8,
	InstruType_MegaSCNeedleDriver :=9,// mega suture-cut needle driver
	InstruType_SCNeedleDriver :=10, // suture-cut needle driver
	InstruType_RoundTipScissors :=11,
	InstruType_ProGraspForceps :=12,
	InstruType_MarylandForceps :=13, // Maryland bipolar forceps
	InstruType_FenestratedForceps :=14, // Fnestrated bipolar forceps
	InstruType_CurvedScissors :=15, // monopolar curved scissors
	InstruType_CauteryHook :=16,
	InstruType_CauterySpatula :=17,
	InstruType_Endoscope := 20,
	InstruType_UltrasoundKnifeS :=42,
	InstruType_UltrasoundKnifeU :=43,
	InstruType_First := InstruType_CadiereForceps,
	InstruType_Last := InstruType_UltrasoundKnifeU
);
END_TYPE

// ---- DUTs/Enum/E_MasterArmState.TcDUT
// Notice: Each state has a corresponding controller, which has a fixed index.
// Add the new state at the end and update the total num
TYPE E_MasterArmState :
(
	MasterArmState_Error := 1,
	MasterArmState_Init :=2,
	MasterArmState_Home :=3,
	MasterArmState_Standby :=4,
	MasterArmState_Matching :=5,
	MasterArmState_Ready :=6,
	MasterArmState_MasterSlave :=7,
	MasterArmState_Clutch :=8,
	MasterArmState_Endoscope :=9,
	MasterArmState_Cart := 10,
	MasterArmState_GravityCali := 11,
	MasterArmState_Test :=12,
	MasterArmState_Disable :=13,
	MasterArmState_Performance :=14,
	
	MasterArmState_totalNum :=MasterArmState_Performance
);
END_TYPE

// ---- DUTs/Enum/E_SlaveArmState.TcDUT
TYPE E_SlaveArmState :
(
	SlaveArmState_Error := 1,
	SlaveArmState_Init :=2,
	SlaveArmState_SelfCheck :=3,
	SlaveArmState_Standby :=4,
	SlaveArmState_MountPanel:=5,
	SlaveArmState_PanelReady :=6,
	SlaveArmState_MountInstru :=7,
	SlaveArmState_InstruReady :=8,
	SlaveArmState_MasterSlave :=9,
	SlaveArmState_ScopeReady :=10,
	SlaveArmState_EndoScope :=11,
	SlaveArmState_Adjust :=12,
	SlaveArmState_Package :=13,
	SlaveArmState_Cart := 14,
	SlaveArmState_GravityCali := 15,
	SlaveArmState_Test := 16,
	SlaveArmState_InstruRetract :=17,
	SlaveArmState_InstruInvasion :=18,
	SlaveArmState_Disable :=19,
	
	SlaveArmState_totalNum :=SlaveArmState_Disable
);
END_TYPE

// ---- DUTs/Structure/MasterSlaveCommunication/ST_MasterStatus.TcDUT
// Output from master arm control task, including arm status and cartesian data
// Input to safety task and Slave controller
TYPE ST_MasterStatus :
STRUCT
	// linear motion scale
	m_motionScale : LREAL:=1.5;
	
	// state machine
	m_armState:ARRAY[1..g_mArmNum] OF E_masterArmState := [2(MasterArmState_Error)];
	
	// index(0 to 4) of slave arm which is tele-linked to master arm
	m_teleSlaveArmIdx :ARRAY[1..g_mArmNum] OF E_MatchedSlaveArmIdx;
	
	// grip angle
	m_gripAngle:ARRAY[1..g_mArmNum] OF LREAL;
	
	// command arm pose in shoulder coordinate
	m_cmdArmPose :ARRAY[1..g_mArmNum] OF ST_Frame;
	
	// current arm pose in shoulder coordinate
	m_curArmPose:ARRAY[1..g_mArmNum] OF ST_Frame;
	
	// command arm twist[linear velocity; angular veloicty] in shoulder coordinate
	m_cmdArmTwist:ARRAY[1..g_mArmNum] OF Vec6d;
	
	// current arm twist[linear velocity; angular veloicty] in shoulder coordinate
	m_curArmTwist:ARRAY[1..g_mArmNum] OF Vec6d;
	
	//self check status
	m_selfCheckStatus : ARRAY [1..g_mArmNum] OF BOOL;
	
	//grip Hall Sensor
	m_gripHallSensor : ARRAY [1..g_mArmNum] OF UDINT;
	
	//slave on line
	m_slaveOnLine : BOOL;
	
	//msater-slave matching status
	m_IKSuccess :ARRAY [1..g_mArmNum] OF BOOL;
	
	//msater-slave matching time
	m_timePeriod :ARRAY [1..g_mArmNum] OF LREAL;
	
	//master arms mapping slave arms
	m_matchedMasterArmIdx : ST_MatchedMasterArmIdx;
END_STRUCT
END_TYPE

// ---- DUTs/Structure/MasterSlaveCommunication/ST_SlaveStatus.TcDUT
// Output from slave arm control task, including arm status and cartesian data
// Input to safety task and Master controller
TYPE ST_SlaveStatus :
STRUCT
	// slave heart beat
	m_slaveHeartBeat :INT:=0;
	
	// slave self-check pass
	m_selfCheckPass :BOOL :=false;
	
	// state machine
	m_armState:ARRAY[1..g_sArmNum] OF E_SlaveArmState:=[g_sArmNum(SlaveArmState_Init)];
	
	// instrument info
	m_instruStauts: ARRAY[1..g_sArmNum] OF ST_InstruStatus;
	
	// flag if endoscope is mounted
	m_endoscopeMounted :BOOL := FALSE;
	
	// endoscope pose in cart coordinate
	m_endoscopePose : ST_Frame;

	// current arm pose in endoscope coordinate
	m_curArmPose:ARRAY[1..g_sArmNum] OF ST_Frame;
	
	// master slave pose error [position, angle*axis] in endoscope coordinate
	m_masterSlavePoseError :ARRAY[1..g_sArmNum] OF Vec6d; 
	
	//slave aseptic deployment complete flag
	m_asepticDeployCompleteFlag : BOOL;
	
	//slave robot stop button trigger
	m_slaveStopButton : BOOL;
END_STRUCT
END_TYPE

// ---- DUTs/Structure/ST_EtherCATState.TcDUT
TYPE ST_EtherCATState :
STRUCT
	EtherCATState : BOOL;
	CRCPortA :UDINT;
	CRCPortB :UDINT;
	CRCPortC :UDINT;
END_STRUCT
END_TYPE

// ---- DUTs/Structure/ST_InstruStatus.TcDUT
TYPE ST_InstruStatus :
STRUCT
	
	m_ready:BOOL := FALSE;
	m_type : E_InstrumentType := InstruType_UNKNOWM;
	m_fingerAngle:LREAL := 0.0;
	m_energyType :UINT :=0;
END_STRUCT
END_TYPE

// ---- DUTs/Structure/ST_MatchedMasterArmIdx.TcDUT
TYPE ST_MatchedMasterArmIdx :
STRUCT
	left1ArmIdx : UINT :=1;
	left2ArmIdx : UINT :=2;
	right1ArmIdx : UINT :=3;
	right2ArmIdx : UINT :=4;
END_STRUCT
END_TYPE

// ---- DUTs/Structure/TasksCommunication/ST_CartUIData.TcDUT
TYPE ST_CartUIData :
STRUCT
	m_ergonomicCrl: ST_ergonCtrlEnable;
	m_cmdErgonomicCrl : ST_ergonomicCtrlData;
	m_cmdCancelErgonPos :Vec4d;
	m_cmdJntPos :Vec4d;
END_STRUCT
END_TYPE

// ---- DUTs/Structure/TasksCommunication/ST_MasterDynaData.TcDUT
TYPE ST_MasterDynaData :
STRUCT
	// mass matrix in joint space
	m_massMat :ARRAY[1..g_mArmNum] OF Mat7d;
	
	// mass matrix in cartesian space
	m_lambda :ARRAY[1..g_mArmNum] OF Mat6d;
	
	// dynamic nullspace
	m_dynaNullspace :ARRAY[1..g_mArmNum] OF Mat7d;
	
	// gravity
	m_gravity :ARRAY[1..g_mArmNum] OF Vec7d;
	
	// friction
	m_friction :ARRAY[1..g_mArmNum] OF Vec7d;
	
	// external torque
	m_jntExtTrq :ARRAY[1..g_mArmNum] OF Vec7d;
END_STRUCT
END_TYPE

// ---- DUTs/Structure/TasksCommunication/ST_MasterUIData.TcDUT
// Output from UI controller
// Input to master arm control task and cart control task  
TYPE ST_MasterUIData :
STRUCT
	m_motionScale:LREAL := 1.5;
	m_selfCheckFlag:BOOL := FALSE;
	m_masterArmDisableFlag :ARRAY[1..2] OF BOOL:=[2(FALSE)];
	m_enableHandClutch :BOOL :=true;
END_STRUCT
END_TYPE

// ---- DUTs/Structure/TasksCommunication/ST_CartStatus.TcDUT
// Output from cart control task
// Input to master arm control task  
TYPE ST_CartStatus :
STRUCT
	m_initFlag :BOOL:= false;
	m_monitorAngle:LREAL := 0.0;
	m_armSwitch:BOOL := FALSE;
	m_clutchSwitch:BOOL := FALSE;
	m_endoscopeSwitch:BOOL := FALSE;
	m_instrumentPowerSwitch:BOOL := FALSE;
	m_surgonReady :BOOL :=false;
	m_consoleInAdjust:BOOL := FALSE;
	m_consoleInManualAdjust:BOOL := FALSE;
	m_ergonAdjustArrival :BOOL;
	m_cancelErgonAdjustArrival :BOOL;
	m_pedalHover : ARRAY [1..2] OF BOOL;
	m_electricKnifePedalTrigger : ARRAY [1..2] OF INT;
END_STRUCT
END_TYPE

// ---- DUTs/Structure/TasksCommunication/ST_MasterJointData.TcDUT
// Output from master arm control task 
// Input to safety task and force controller task
TYPE ST_MasterJointData :
STRUCT
	// joint position compute with motor encoder
	m_curMotorPos :ARRAY[1..g_mArmNum] OF Vec7d;
	
	// joint position compute with link/abs encoder
	m_curLinkPos :ARRAY[1..g_mArmNum] OF Vec7d;
	
	// target joint position 
	m_cmdJntPos :ARRAY[1..g_mArmNum] OF Vec7d;
	
	// current joint position 
	m_curJntPos :ARRAY[1..g_mArmNum] OF Vec7d;
	
	// target joint velocity 
	m_cmdJntVel :ARRAY[1..g_mArmNum] OF Vec7d;
	
	// current joint position 
	m_curJntVel :ARRAY[1..g_mArmNum] OF Vec7d;
	
	// command joint torque 
	m_cmdJntTrq :ARRAY[1..g_mArmNum] OF Vec7d;
	
	// current joint torque 
	m_curJntTrq :ARRAY[1..g_mArmNum] OF Vec7d;
	
	// raw joint current  
	m_rawJntCurrent :ARRAY[1..g_mArmNum] OF Vec7d;
	
	// filtd  joint current  
	m_filtJntCurrent :ARRAY[1..g_mArmNum] OF Vec7d;
	
	// command joint current 
	m_cmdJntCurrent :ARRAY[1..g_mArmNum] OF Vec7d;
END_STRUCT
END_TYPE

// ---- DUTs/Structure/TasksCommunication/ST_MotorOutputs.TcDUT
TYPE ST_MotorOutputs :
STRUCT
	// driver control word
	m_controlWord: UINT :=DriverCtrlWord_INIT;
	
	// motor control mode, 0 for position mode, 1 for torque mode
	m_opMode : SINT :=INT_TO_SINT(DriverOPMode_Pos);;
	
	// target motor encoder
	m_cmdMotorEncoder :DINT := 0;
	
	// motor current to IO
	m_cmdCurrent :DINT := 0;
	
END_STRUCT
END_TYPE

// ---- DUTs/Structure/TasksCommunication/ST_SlaveJointData.TcDUT
TYPE ST_SlaveJointData :
STRUCT
	// joint position compute with motor encoder
	m_curMotorPos :ARRAY[1..g_sArmNum] OF Vec8d;
	
	// joint position compute with link/abs encoder
	m_curLinkPos :ARRAY[1..g_sArmNum] OF Vec8d;
	
	// target joint position 
	m_cmdJntPos :ARRAY[1..g_sArmNum] OF Vec8d;
	
	// current joint position 
	m_curJntPos :ARRAY[1..g_sArmNum] OF Vec8d;
	
	// target joint velocity 
	m_cmdJntVel :ARRAY[1..g_sArmNum] OF Vec8d;
	
	// current joint position 
	m_curJntVel :ARRAY[1..g_sArmNum] OF Vec8d;
	
	// command joint torque 
	m_cmdJntTrq :ARRAY[1..g_sArmNum] OF Vec8d;
	
	// current joint torque 
	m_curJntTrq :ARRAY[1..g_sArmNum] OF Vec8d;
	
	// raw joint current  
	m_rawJntCurrent :ARRAY[1..g_sArmNum] OF Vec8d;
	
	// filtd  joint current  
	m_filtJntCurrent :ARRAY[1..g_sArmNum] OF Vec8d;
	
	// command joint current 
	m_cmdJntCurrent :ARRAY[1..g_sArmNum] OF Vec8d;
END_STRUCT
END_TYPE

// ---- DUTs/Structure/TasksCommunication/ST_SafetyData.TcDUT
// Output from safety check task
// Input to master arm control task
TYPE ST_SafetyData :
STRUCT
	m_masterErrFlag :ARRAY[1..g_mArmNum] OF BOOL :=[2(FALSE)];
	m_cartErrFlag :Vec4b :=[4(FALSE)];
END_STRUCT
END_TYPE

// ---- DUTs/Structure/ST_MasterInputDataPool.TcDUT
// Struct contains all data from other tasks and controller used for master control
TYPE ST_MasterInputDataPool :
STRUCT
		
	// UI information, import from UI controller
	m_UIData :ST_MasterUIData;
	
	// safety information, import from safety check task
	m_safetyData AT %I*: ST_SafetyData;
	
	// cart information, import from other task
	m_cartStatus AT %I*:ST_CartStatus;
	
	// slave robot status, copy from MSCommu_SlaveStauts
	m_slaveStatus :ST_SlaveStatus;
	
	// master dynamic data
	m_masterDynaData AT %I* : ST_MasterDynaData;
	
END_STRUCT
END_TYPE

// ---- DUTs/Structure/TasksCommunication/ST_CartJointData.TcDUT
TYPE ST_CartJointData :
STRUCT
	// joint position compute with motor encoder
	m_curMotorPos : Vec4d;
	
	// joint position compute with link/abs encoder
	m_curLinkPos : Vec4d;
	
	// target joint position 
	m_cmdJntPos : Vec4d;
	
	// current joint position 
	m_curJntPos : Vec4d;
	
	// target joint velocity 
	m_cmdJntVel : Vec4d;
	
	// current joint position 
	m_curJntVel : Vec4d;
	
	// command joint torque 
	m_cmdJntTrq : Vec4d;
	
	// current joint torque 
	m_curJntTrq : Vec4d;
	
	// raw joint current  
	m_rawJntCurrent : Vec4d;
	
	// filtd  joint current  
	m_filtJntCurrent : Vec4d;
	
	// command joint current 
	m_cmdJntCurrent : Vec4d;
END_STRUCT
END_TYPE

// ---- DUTs/Structure/UICommunication/ST_arm_distribution.TcDUT
TYPE ST_arm_distribution :
STRUCT
	//slave arm 1 mapping left arm or right arm
	m_arm1InLeftOrRight : UINT;
	
	//slave arm 2 mapping left arm or right arm
	m_arm2InLeftOrRight : UINT;
	
	//slave arm 3 mapping left arm or right arm
	m_arm3InLeftOrRight : UINT;
	
	//slave arm 4 mapping left arm or right arm
	m_arm4InLeftOrRight : UINT;
	
	m_leftMappingSlaveArm : ARRAY [1..2] OF UINT:=[1,2];
	m_rightMappingSlaveArm : ARRAY [1..2] OF UINT:=[3,4];
END_STRUCT
END_TYPE

// ---- DUTs/Structure/UICommunication/ST_ergonCtrlEnable.TcDUT
TYPE ST_ergonCtrlEnable :
STRUCT
	//recovery ergonomics enable 
	m_recovErgonEnable : BOOL;

	//recovery ergonomics finshed
	m_recovErgonFinshed : BOOL;
	
	//cancel recovery ergonomics enable 
	m_cancelRecovErgonEnable : BOOL;
	
	//cancel recovery ergonomics finshed
	m_cancelRecovErgonFinshed : BOOL;
	
	//ergonomics information modify
	m_ergonInfoModify : BOOL;

END_STRUCT
END_TYPE

// ---- DUTs/Structure/UICommunication/ST_ergonomicCtrlData.TcDUT
TYPE ST_ergonomicCtrlData :
STRUCT
	m_monitorHeight : REAL;
	m_headAngle : REAL;
	m_handrailHeight : REAL;
	m_footDistance : REAL;
END_STRUCT
END_TYPE

// ---- DUTs/Structure/UICommunication/ST_instrument_info.TcDUT
TYPE ST_instrument_info :
STRUCT
	is_connected:BOOL;  //器械已连接
	is_ready:BOOL;  //器械正常
	clamp_match:BOOL;  //器械主从匹配状态
	master_slave_state:BOOL;  //器械主从状态，是否有主从关系
	is_energy:BOOL;
	is_bipolar:BOOL;
	is_available: BOOL;
	is_active:BOOL;
	is_hover:BOOL;
	pedal_active:UINT;
	
	id:UINT;
	hand_signs:UINT;
	total_lilfe:UINT;
	remain_life:UINT;
	dof_map:ARRAY[1..5] OF UINT;
	
	size:REAL;
	range_min:ARRAY[1..5] OF REAL;
	range_max:ARRAY[1..5] OF REAL;
	torque_max:ARRAY[1..5] OF REAL;
	ratio:ARRAY[1..5] OF REAL;

	name:STRING;
	type_1:STRING;
	serial_number:STRING;
	path:STRING;	
END_STRUCT
END_TYPE

// ---- DUTs/Structure/UICommunication/ST_scope_info.TcDUT
TYPE ST_scope_info :
STRUCT
	is_connected:BOOL;
	is_ready:BOOL;
	id:UINT;
	scope_deg:UINT;
	scope_up_down:UINT;
	scope_gravity_angle:UINT;
	scope_name:STRING;
END_STRUCT
END_TYPE

// ---- DUTs/Type/Vec7b.TcDUT
TYPE Vec7b : ARRAY[1..7] OF BOOl; END_TYPE

// ---- DUTs/Type/Mat34.TcDUT
TYPE Mat34 : ARRAY[1..3, 1..4] OF LREAL; END_TYPE

// ---- DUTs/Type/Mat37.TcDUT
TYPE Mat37 : ARRAY[1..3, 1..7] OF LREAL; END_TYPE

// ---- DUTs/Type/Mat43.TcDUT
TYPE Mat43 : ARRAY[1..4, 1..3] OF LREAL; END_TYPE

// ---- DUTs/Type/Mat4d.TcDUT
TYPE Mat4d : ARRAY[1..4, 1..4] OF LREAL; END_TYPE

// ---- DUTs/Type/Mat5d.TcDUT
TYPE Mat5d : ARRAY[1..5, 1..5] OF LREAL; END_TYPE

// ---- DUTs/Type/Vec4d.TcDUT
TYPE Vec4d : ARRAY[1..4] OF LREAL; END_TYPE

// ---- DUTs/Type/Vec4i.TcDUT
TYPE Vec4i : ARRAY[1..4] OF INT; END_TYPE

// ---- DUTs/Type/Vec6i.TcDUT
TYPE Vec6i : ARRAY[1..6] OF INT; END_TYPE

// ---- DUTs/Type/Vec4b.TcDUT
TYPE Vec4b : ARRAY[1..4] OF BOOl; END_TYPE

// ---- DUTs/Type/Vec7di.TcDUT
TYPE Vec7di : ARRAY[1..7] OF DINT; END_TYPE

// ---- DUTs/Type/Vec8d.TcDUT
TYPE Vec8d : ARRAY[1..8] OF LREAL; END_TYPE

// ---- DUTs/Enum/E_DriverOPMode.TcDUT
TYPE E_DriverOPMode :
(
	DriverOPMode_Pos := 0, // driver position control
	DriverOPMode_Trq :=1, // driver torque control, robot force control
	DriverOPMode_PosTrq :=2 // driver torque control, robot position contorl
);
END_TYPE

// ---- DUTs/Type/Vec7d.TcDUT
TYPE Vec7d : ARRAY[1..7] OF LREAL; END_TYPE

// ---- DUTs/Type/Vec7i.TcDUT
TYPE Vec7i : ARRAY[1..7] OF INT; END_TYPE

// ---- SafetyCheck/safetyCheckDUT/checkDelay.TcDUT
TYPE checkDelay  :
STRUCT
	T_armJntEncErr:ARRAY [1..7] OF FB_TON;
	T_driveErr:ARRAY [1..7] OF FB_TON;
	T_linkEncErr:ARRAY [1..7] OF FB_TON;
	T_jntStatusErr:ARRAY [1..7] OF FB_TON;
	T_currentIsNotUpdate:ARRAY [1..7] OF FB_TON;
	T_outOfLimit:ARRAY [1..7] OF TON;
	T_armJntFollowErr:ARRAY [1..7] OF FB_TON;
	T_jntVelErr:ARRAY [1..7] OF FB_TON;
	T_jntCurrentErr:ARRAY [1..7] OF FB_TON;
	T_spacePoseErr:ARRAY [1..7] OF FB_TON;
	
	T_cartJntEncErr:ARRAY [1..4] OF FB_TON;
	T_cartDriveErr:ARRAY [1..4] OF FB_TON;
	T_cartLinkEncErr:ARRAY [1..4] OF FB_TON;
	T_cartJntStatusErr:ARRAY [1..4] OF FB_TON;
	T_cartCurrentIsNotUpdate:ARRAY [1..4] OF FB_TON;
	T_cartOutOfLimit:ARRAY [1..4] OF FB_TON;
	T_cartJntFollowErr:ARRAY [1..4] OF FB_TON;
	T_cartJntVelErr:ARRAY [1..4] OF FB_TON;
	T_cartJntCurrentErr:ARRAY [1..4] OF FB_TON;
END_STRUCT
END_TYPE

// ---- SafetyCheck/safetyCheckDUT/checkDelayTime.TcDUT
TYPE checkDelayTime :
STRUCT
	//motor encoder and joint encoder deviation delay time
	Ti_armJntEncErr:TIME:=T#0.1S;
	//drive error delay time
	Ti_driveErr:TIME:=T#0.1S;
	//joint encoder ununuited delay time
	Ti_linkEncErr:TIME:=T#5S;
	//joint status error delay time 
	Ti_jntStatusErr:TIME:=T#1S;
	//motor current is not update delay time
	Ti_currentIsNotUpdate:TIME:=T#20S;
	//joint postion out of limit
	Ti_outOfLimit:TIME:=T#0.1S;
	//joint follow error delay time
	Ti_armJntFollowErr:TIME:=T#0.1S;
	//joint vel error delay time
	Ti_jntVelErr:TIME:=T#0.05S;
	//joint current error  delay time
	Ti_jntCurrentErr:TIME:=T#0.1S;
	//space pose error  delay time
	Ti_spacePoseErr:TIME:=T#0.1S;

	
	Ti_carDualEncDev:TIME:=T#0.02S;
	Ti_carDriveErr:TIME:=T#1S;
	Ti_carActSec:TIME:=T#10S;
	Ti_carJntStatus:TIME:=T#1S;
	Ti_carTorMotor:TIME:=T#20S;
	Ti_caroutofLimit:TIME:=T#0.1S;
	Ti_carFollowDev:TIME:=T#0.02S;
	Ti_carJntVel:TIME:=T#0.05S;
	Ti_carJntCurrent:TIME:=T#1S;
END_STRUCT
END_TYPE

// ---- SafetyCheck/safetyCheckDUT/checkInputVariable.TcDUT
TYPE checkInputVariable :
STRUCT
	EmergencyStop:BOOL;
	m_cartDriverInput :ARRAY[1..g_maxCartJoint] OF ST_MotorInputs; 
	m_cartDriverOutput :ARRAY[1..g_maxCartJoint] OF ST_MotorOutputs;
	m_masterDriverInput :ARRAY[1..g_mJntNum] OF ST_MotorInputs; 
	m_masterDriverOutput :ARRAY[1..g_mJntNum] OF ST_MotorOutputs;
	m_motorCurrentIntegral : vec7d;
	m_motorEncSaltaValue : ARRAY[1..g_mJntNum] OF DINT;
	m_EtherCATState:ARRAY [1..g_maxArmJoint] OF ST_EtherCATState;		
	m_spacePoseErr: vec6d;
	m_promptStatus:ARRAY [1..20] OF BOOL;
	m_promptLocation:ARRAY [1..20] OF UDINT;
	m_selfCheckFail : BOOL;
	
	SlaveStopButton:BOOL;
	PCStopButton :UINT;
	MasterStopButton :BOOL;
	
	m_cartEtherCATState:ARRAY [1..g_maxCartJoint] OF ST_EtherCATState;
END_STRUCT
END_TYPE

// ---- SafetyCheck/safetyCheckDUT/checkPermit.TcDUT
TYPE checkPermit :
STRUCT
	m_armJntEncErr :vec7b;
	m_driveErr :vec7b;
	m_jntStatusErr :vec7b;
	m_currentIsNotUpdate :vec7b;
	m_linkEncErr :vec7b;
	m_motPhieErr:vec7b;
	m_outOfLimit :vec7b;
	m_armJntFollowErr :vec7b;
	m_jntVelErr :vec7b;
	m_jntCurrentErr :vec7b;
	m_cmdJntSaltation:vec7b;
	m_spacePoseErr:vec7b;
	

	m_cartJntStatus : vec4b:=[4(TRUE)];
	m_cartCurrentIsNotUpdate : vec4b:=[4(TRUE)];
	m_cartLinkEncErr : vec4b:=[4(TRUE)];
	m_cartDriveErr : vec4b:=[4(TRUE)];
	m_cartJntEncErr : vec4b:=[4(TRUE)];
	m_cartOutOfLimit : vec4b:=[4(TRUE)];
	m_cartFollowErr : vec4b:=[4(TRUE)];
	m_cartJntVelErr : vec4b:=[4(TRUE)];
	m_cartJntCurrentErr : vec4b:=[4(FALSE)];
END_STRUCT
END_TYPE

// ---- SafetyCheck/safetyCheckDUT/ST_Buffer.TcDUT
TYPE ST_Buffer :
STRUCT
	bFull 		: BOOL;
	sPath		: STRING;
	aBuffer 	: ARRAY[0..MAX_CSV_ROWS ] OF ARRAY [0..MAX_CSV_COLUMNS] OF STRING(MAX_CSV_FIELD_LENGTH) ;
	bBuffer 	: ARRAY[0..MAX_CSV_ROWS ] OF ARRAY [0..MAX_CSV_COLUMNS] OF STRING(MAX_CSV_FIELD_LENGTH) ;
	fbWriter 	: FB_Writer;
END_STRUCT
END_TYPE

// ---- SafetyCheck/safetyCheckDUT/T_Buffer.TcDUT
TYPE T_Buffer: ARRAY[ 0..MAX_CSV_ROWS ] OF ARRAY [0..MAX_CSV_COLUMNS] OF STRING(MAX_CSV_FIELD_LENGTH); (* [] (* TODESC *) *)
END_TYPE

// ---- GVLs/Arms/GVL_ArmDynamics.TcGVL
{attribute 'global_init_slot' := '49992'}
{attribute 'qualified_only'}
// Robot3 Data
VAR_GLOBAL CONSTANT
	// arm gravity parameters
	(*graParam=[ 2.7244*m3 + 2.7244*m4 + 2.7244*m5 + 2.7244*m6 + 9.8*mx2 + 9.8*mx9,
				9.8*my2 + 9.8*my9,
				3.577*m4 + 3.577*m5 + 3.577*m6 + 0.49*m9 + 9.8*mx3 + 9.8*mx8
				1.5827*m4 + 1.5827*m5 + 1.5827*m6 + 9.8*my3 + 9.8*my8 + 9.8*mz4
				mz5-my4,	my5+mz6,  	mx4,   	mx5, 	mx6,   	my6
				preF2,   k2,   preF3,    k3,    preF5   k5]*)
	g_gravityParam :ARRAY[1..2, 1..16] OF REAL := 
		[ 6.2624762, -0.0007155225, 3.1411762, 0.48504608, -0.03459308, 0.025676297, 0.0000375, 0.0000351, -0.00001, -0.01593742,
		  7.7845001, 3195.0, 7.7845, 1902.6574, 2.5056201, 481.81768,
		  5.8820792, -0.0002385075, 2.9722568, 0.54387185, -0.037805167, 0.019637397, 0.000012500001, 0.0000117, -0.0000099999999, -0.013195626, 
		  10.732782, 2910.6441, 15.50438, 1786.0662, 2.1109713, 393.46033];
			
	// gravity deviation
	g_gravityDeviaion :ARRAY[1..2, 1..7] OF REAL :=
	[ 0.0, 0.0, 0.0, 0.0, 0.0, 0.0, 0.0, 
	 0.0, 0.0, 0.0, 0.0, 0.0, 0.0, 0.0];
	  
	// arm friction parameters [a1,b1,...a7,b7];
	// friction = a * gravity + b; only joint 5 and 6 is identified
	g_jntFrictionParam :ARRAY[1..2, 1..4] OF LREAL :=
	[ 0.18558566, 0.013430012, 0.1933446, 0.0056009337,
	  0.25838222, 0.0080955163, 0.3329508, 0.0062479093];
	g_maxJntFriction : Vec7d :=[0, 0, 0, 0, 0.05, 0.05, 0];
	
	//################ dynamic reference model parameters below ###########################
	// link mass [m1, m2, m3, m4, m5, m6, m7, m8, m9]
	g_linkMass :ARRAY[1..9] OF LREAL :=[2.676, 0.825, 0.547, 0.25, 0.195, 0.194, 0.05, 0.111, 0.09] ;
	
	// lin center of amss
	g_linkCOM :ARRAY[1..9,1..3] OF LREAL := [   1.376E-3,    -1.019E-3,  -81.464E-3,
										   90.622E-3,   -0.113E-3,  15.088E-3,
										   167.4E-3,    3.7E-3,     -0.438E-3,
										   0.1E-3,      98.49E-3,   -55.74E-3,
										   0.12E-3,     76.667E-3,  -36E-3,
										   0,           -61.63E-3,  27.3E-3,
										   0.06E-3,     -0.08E-3,   17.671E-3,
										   11E-3,       -3.364E-3,  39.265E-3,
										   143e-3,      0.495e-3,   24.253e-3];
	// link  inertial
    // [Ixx,Iyy,Izz, Ixy,Ixz, Iyz]
 	g_linkInertia :ARRAY[1..9,1..6] OF LREAL :=[  19.63E-3,   16.43E-3,  12.7E-3,   -0.3222E-3,    -0.667E-3,     -0.0268E-3,
												   1.017E-3,   6.637E-3,  5.935E-3,  -0.037E-3,     -0.238E-3,     0.06E-3,
												   0.161E-3,   9.572E-3,  9.586E-3,  0.0447E-3,     0.0277E-3,     0.465E-6,
												   0.992E-3,   0.707E-3,  0.335E-3,  0.2E-6,     2E-6,       0.224E-3,
												   0.402E-3,   0.25E-3,   0.186E-3,  0.002E-6,   -1.2E-6,    0.106E-3,
												   0.281E-3,   0.178E-3,  0.137E-3,  0.076E-6,   0.09E-6,    0.056E-3,
												   0.0255E-3,  0.0259E-3, 5.96E-6,0.34E-6,    -3E-9,      24E-9,
												   0.033E-3,   0.0976E-3, 0.126E-3,  3E-6,       -5E-6,      -0.162E-6,
												   4.9E-6,  0.757E-3,  0.760E-3,  2.6E-6,     -5.3E-6,    -18E-9];

	//################ DO NOT modify parameters below ###########################
	//  motor inertial at link size
	g_motorInertia :ARRAY[1..7] OF LREAL := [34.7E-7, 34.7E-7, 34.7E-7, 9.26E-7, 0.495E-7, 0.495E-7, 0.495E-7];
	
	// spring parameters
	// spring2 [L0, b1, b2, l1, r0]
	g_spring2Param :ARRAY[1..5] OF LREAL :=[101.6E-3, 14.5E-3, 15E-3, 172E-3, 31E-3];
	// spring3 [L0, b1, b2, l1, r0,d]
	g_spring3Param :ARRAY[1..6] OF LREAL :=[101.6E-3, 14E-3, 15E-3, 172E-3, 30E-3, 10E-3];
	// spring5 [L0, s1, L1, r0, beta]
	g_spring5Param :ARRAY[1..5] OF LREAL :=[34.93E-3, 34.3E-3, 100E-3, 12.5E-3, 32.02*g_deg2rad];
	
END_VAR

// ---- GVLs/Arms/GVL_ArmJointCaliData.TcGVL
{attribute 'qualified_only'}
// Robot3 Data
VAR_GLOBAL CONSTANT									 
	// absolute encoder value at minimal joint positon
	g_minLinkEncoder :ARRAY[1..g_mArmNum, 1..g_mJntNum] OF DINT :=
		[5320292, 1637888, 16267012, 9121008, 16329376, 6965264, 0,
		 54048, 5138400, 12480240, 3380960, 9526944, 5270880, 0];
		 
	// absolute encoder value at maximum joint positon
	g_maxLinkEncoder :ARRAY[1..g_mArmNum, 1..g_mJntNum] OF DINT :=
		[16734116, 13586832, 3813732, 14235024, 11133568, 11256240, 0,
		 11534296, 16020072, 96940, 8157232, 13636784, 5270880, 0];
	
	// absolute encoder value at calibrated positon
	g_caliLinkEncoder :ARRAY[1..g_mArmNum, 1..g_mJntNum] OF DINT :=
		[2383568, 16504180, 1064304, 2073472, 6104944, 9016224, 13420592,
		 14507208, 2154776, 14028284, 15460608, 3197104, 7324448, 14964448];
	
	 // if absolute encoder value cross zeros within joint motion range
	 // NOTICE: joint 7 is always 0.
	g_linkEncZeroCross :ARRAY[1..g_mArmNum, 1..g_mJntNum] OF INT :=
		[1, 1, 1, 1, 1, 0, 1,
		 1, 1, 1, 1, 1, 0, 1];
		 
	// limit value of gripper hall sensor
	g_minHallSensorValue :ARRAY[1..2] OF DINT:=[2687067,3145824];
	g_maxHallSensorValue :ARRAY[1..2] OF DINT  :=[34800091,36635182];
		 
 	//################ DO NOT modify parameters below ###########################	
	// abolute encoder expanded limit buffer in case there is calibrtion error at limit position
	g_linkEncLimitBuffer : DINT := 100000;
	
	// flag if joint can rotate multiple cycles
	g_multipleCyclesJoint :ARRAY[1..g_mArmNum, 1..g_mJntNum] OF INT :=
		[0, 0, 0, 0, 0, 0, 1,
		 0, 0, 0, 0, 0, 0, 1];
		 
	// joint position at link encoder calibrated point
	g_linkEncCaliJntPos :ARRAY[1..g_mArmNum, 1..g_mJntNum] OF LREAL :=
		[0.0, -PI/2, 0.0, -pi, pi, -PI/2, 0.0,
		 0.0, -PI/2, 0.0, 0.0, pi, PI/2, 0.0];

END_VAR

// ---- GVLs/Arms/GVL_ArmKinematic.TcGVL
// use slot attribute larger than 49990, which is the default one, if it depends on variable in other file
{attribute 'global_init_slot' := '49991'} 
VAR_GLOBAL CONSTANT 

// distance between shoulders of left and right arm
g_shoulderDistance :LREAL := 0.5;

// master arm shoulder rotation in base monitor pose(0 rotate angle)
g_shoulderRotInMonitor : Mat3d :=[0.0,	-1.0,	0.0,
								  0.0,	0.0,	1.0,
								  -1.0,	0.0,	0.0];
 	
(* 
% DH definetion
% !!!!NOTE: q4 is the DH joint position, NOT the motor one
% paramters definiton:
% d1: arm origin to joint1 
% a3: upper arm length
% a4: lower arm length
% d4: wrist height
% a9: parallel structure width
% DH definition:
% index     parent  alpha   a       theta   d       active
% 1         0       0       0       q1      d1      1
% 2         1       -90     0       q2      0       1
% 3         0       0       a3      q3      0       0
% 4         3       -90     a4      q4      d4      1
% 5         4       90      0       q5      0       1
% 6         5       -90     0       q6      0       1
% 7         6       90      0       q7      0       1

% 8         1       -90     0       q8      0       1
% 9         8       0       a9      q9      0       0
% 10        9       0       a3      q10     0       0
% 11        3       0       a9      0       0       fixed

%q4 = motor_q4+q8-q2-90
%q3 = q8 - q2;
%q9 = q2-q8;
%q10 = q8-q2

*)
g_d1:LREAL:=0.26085;
g_d4:LREAL:=0.1615;
g_a3:LREAL:=0.278;
g_a4:LREAL:=0.365;
g_a9:LREAL:=0.06;

//alpha,a,d,theta	
g_masterArmDH:ARRAY[1..9,1..4] OF LREAL :=[0,	0,		g_d1,	0,      
										-pi/2,	0,		0,		0,
										0,		g_a3,	0,		0,
										-pi/2,	g_a4,	g_d4,	0,       
										pi/2,	0,		0,		0,
										-pi/2,	0,		0,		0,
										pi/2,	0,		0,		0,
										-pi/2,	0,		0,		0,// joint 8
										0,		g_a9, 	0,		0];
											
// master grip angle fitting coefficients(wrt normalized hall sensor value)
g_masterGripAngleFitCoeff : ARRAY[1..6] OF LREAL :=
	[-2.767665451, 8.744429877, -10.74377687, 6.69841, -2.449592087, 0.5188884865];
g_maxGripAngle : LREAL := 30.0 * g_deg2Rad;
g_minGripAngle :LREAL  := 0.0;

END_VAR

// ---- GVLs/Arms/GVL_ControlParameters.TcGVL
{attribute 'global_init_slot' := '49991'}
VAR_GLOBAL CONSTANT
	// master arm joint position controller parameters
	g_posKp :ARRAY[1..7] OF LREAL :=[0.0, 0.0, 0.0, 4.0, 2.0, 1.0, 0.5];
	g_posKd :ARRAY[1..7] OF LREAL :=[0.0, 0.0, 0.0, 0.1, 0.035, 0.05, 0.01];
	g_posKi :ARRAY[1..7] OF LREAL :=[0.0, 0.0, 0.0, 20.0, 10.0, 10.0, 5.0];
	g_posKiLimit :ARRAY[1..7] OF LREAL :=[500,500,500,500,100,100,100];// define in current
	g_posCtrlLimit :ARRAY[1..7] OF LREAL :=[1000,1000,1000,1000,300,200,200];// define in current
	
	// redundant joint4 following motion parameters
	g_jnt4MaxFollowVel :LREAL :=2*pi;
	g_jnt4MaxFollowAcc :LREAL :=6*pi;
	
	// control tolerance
	g_jntCtrlAngTolLow :LREAL :=0.2*g_deg2Rad;
	g_jntCtrlAngTolHigh :LREAL :=1.0*g_deg2Rad;
	g_cartCtrlPosTol :LREAL :=0.0002;
	g_cartCtrlOriTol :LREAL :=0.2*g_deg2Rad;
	
	// filter cut-off frequency for master grip angle
	g_gripAngLpfCutoffFreq :LREAL := 20;
	
	// filter cut-off frequency for velocity and torque
	g_curJntVelLpfCutoffFreq :LREAL := 30;
	g_cmdJntPosLpfCutoffFreq :LREAL := 30;
	g_curJntTrqLpfCutoffFreq :LREAL := 300;
	g_cmdJntTrqLpfCutoffFreq :LREAL := 300;
	
	// controller would keep command unchanged when error 
	// between command and current value is less than this value
	g_jntCtrlErrForCmdHold :LREAL :=2.0*g_deg2Rad;
	
	// joint is assumed to be static if velocity is less than this value
	g_jntStaticVelThres :LREAL :=0.2*g_deg2Rad;
	
	// home motion parameters
	g_homePosture:ARRAY [1..2, 1..7] OF LREAL:=[0.0, -PI/2, 0, -PI, PI, -PI/2, 0,
							 			  			0.0, -PI/2, 0, 0, PI, PI/2, 0];
	g_homeMaxjntVel:Vec7d:=[1.0, 1.0, 1.0, 1.0, 1.0, 1.0, 1.0];
	g_homeMaxjntAcc:Vec7d:=[1.0, 1.0, 1.0, 2.0, 2.0, 2.0, 2.0];
	g_homeMaxjntJerk:Vec7d:=[7(4.0)];
	
	 // joint observer paramters
	g_jntObvParamL1 :Vec7d :=[0, 0, 0, 0, 300, 300, 0];
	g_jntObvParamL2 :Vec7d :=[0, 0, 0, 0, 1000, 1000, 0];
	g_jntObvParamL3 :Vec7d :=[0, 0, 0, 0, 1000, 1000, 0];
	g_jntObvDamp:Vec7d := [0.8,    0.8,    0.8,     0.05, 0.05, 0.05, 0.05];// TODO: need to be identified
END_VAR

// ---- GVLs/Arms/GVL_ArmJointParameters.TcGVL
{attribute 'global_init_slot' := '49991'}
{attribute 'qualified_only'}
VAR_GLOBAL CONSTANT
	// encoder resolution
	g_incEncoderRes :ARRAY[1..7] OF DINT :=[7(65536)];
	g_absEncoderRes :ARRAY[1..7] OF DINT :=[7(16777216)];
	
	// reduction ratio
	g_motorReduction :ARRAY[1..7] OF LREAL :=[43.9658,26.859,26.8018,(66.0/10)*3,4554.0/130, 4554.0/130,5625.0/361];
	g_absEncoderReduction :ARRAY[1..7] OF LREAL :=[7(1.0)];
	
	// motor parameters
	g_motorTrqConst :ARRAY[1..7] OF LREAL :=[0.0538,0.0538,0.0538,0.0299,0.0193,0.0193,0.0193];
	g_motorMaxCurrent :ARRAY[1..7] OF LREAL :=[1000,1000,1000,1000,300,200,220];//mA
	g_jntMaxTrq :ARRAY[1..7] OF LREAL :=[g_motorMaxCurrent[1]*g_motorReduction[1]*g_motorTrqConst[1]/1000.0,  g_motorMaxCurrent[2]*g_motorReduction[2]*g_motorTrqConst[2]/1000.0,
									g_motorMaxCurrent[3]*g_motorReduction[3]*g_motorTrqConst[3]/1000.0,		g_motorMaxCurrent[4]*g_motorReduction[4]*g_motorTrqConst[4]/1000.0,
									g_motorMaxCurrent[5]*g_motorReduction[5]*g_motorTrqConst[5]/1000.0,		g_motorMaxCurrent[6]*g_motorReduction[6]*g_motorTrqConst[6]/1000.0,
									g_motorMaxCurrent[7]*g_motorReduction[7]*g_motorTrqConst[7]/1000.0];
	
	// motor and absEncoder direction
	g_motorDir :ARRAY[1..2, 1..7] OF INT :=[1, 1, -1, 1, 1, -1, -1,	
											1, 1, -1, 1, 1, -1, -1];
	g_asbEncoderDir :ARRAY[1..2, 1..7] OF INT :=[-1, -1, 1, -1, 1, 1, 1,
												 -1, -1, 1, -1, 1, 1, 1];
																 
	// joint position limit
	//TODO: joint7 is given a large limit for initialization moiton
	//NOTE: joint 4 position is coupled with joint 2/3, so the limit is described by link side
	g_minJntPos: ARRAY[1..2,1..7] OF LREAL:=[-60*g_deg2Rad,	-45*g_deg2Rad-pi/2,		-45*g_deg2Rad, 	-pi/2-220*g_deg2Rad, 	-135*g_deg2Rad+pi,		-45*g_deg2Rad-pi/2,		-330*g_deg2Rad,
											 -60*g_deg2Rad,	-45*g_deg2Rad-pi/2,		-45*g_deg2Rad,	-pi/2+5*g_deg2Rad,		-135*g_deg2Rad+pi,		-45*g_deg2Rad+pi/2,	-330*g_deg2Rad];
	g_maxJntPos: ARRAY[1..2,1..7] OF LREAL:=[60*g_deg2Rad,	60*g_deg2Rad-pi/2,		60*g_deg2Rad,		-pi/2-5*g_deg2Rad,			135*g_deg2Rad+pi,		45*g_deg2Rad-pi/2,		330*g_deg2Rad,
								             60*g_deg2Rad,	60*g_deg2Rad-pi/2,		60*g_deg2Rad,		-pi/2+220*g_deg2Rad,			135*g_deg2Rad+pi,		45*g_deg2Rad+pi/2,		330*g_deg2Rad];
	
	// joint velocity limit
	g_maxJntVel :ARRAY[1..7] OF LREAL :=[7(2*pi)];
	
END_VAR

// ---- GVLs/Cart/GVL_CartJointCaliData.TcGVL
{attribute 'qualified_only'}
// Robot3 Data
VAR_GLOBAL CONSTANT
	(* cart joints are defiend in sequence as below
	[monitor lift, monitor rotate, armset, pedal] *)

	// absolute encoder value at minimal joint positon
	g_minLinkEncoder :ARRAY[1..4] OF DINT :=[10551943, 13637932, 8646306,11744290];
		 
	// absolute encoder value at maximum joint positon
	g_maxLinkEncoder :ARRAY[1..4] OF DINT :=[9057645, 16333724,7704162,10974938];
	
	// absolute encoder value at calibrated positon
	g_caliLinkEncoder :ARRAY[1..4] OF DINT :=[10551943, 13637932, 8646306,11744290];
	
	// if absolute encoder value cross zeros within joint motion range
	g_linkEncZeroCross :ARRAY[1..4] OF INT :=[0, 0, 0, 0];
		
	 //################ DO NOT modify parameters below ###########################
	// abolute encoder expanded limit buffer in case there is calibrtion error at limit position
	g_linkEncLimitBuffer : DINT := 100000;
	
	// flag if joint can rotate multiple cycles
	g_multipleCyclesJoint :ARRAY[1..4] OF INT :=[0, 0, 0, 0];
		 
	// joint position at link encoder calibrated point
	//TODO: joint2 calibration position need to be checked
	g_linkEncCaliJntPos :ARRAY[1..4] OF LREAL :=[0, 0*g_deg2Rad,0,0];

END_VAR

// ---- GVLs/Cart/GVL_CartJointParameters.TcGVL
{attribute 'global_init_slot' := '49991'}
{attribute 'qualified_only'}
VAR_GLOBAL CONSTANT
	(* cart joints are defiend in sequence as below
	[monitor lift, monitor rotate, armset, pedal] *)
	
	// encoder resolution
	g_incEncoderRes :ARRAY[1..4] OF DINT :=[4(65536)];
	g_absEncoderRes :ARRAY[1..4] OF DINT :=[4(16777216)];
	
	// reduction ratio
	g_motorReduction :ARRAY[1..4] OF LREAL :=[2*pi/0.0004682,3317.76,2*pi/0.0004682,1.5*138.0/5*2*pi/0.004];
	// TODO: need to be verified, especially joint2
	g_absEncoderReduction :ARRAY[1..4] OF LREAL :=[1.534, 1 , 1.534, 1.534];// 2*pi/(reduction*g_absEncoderRes)=Line_Resolution_car(from old code, 0.001*2/2^13)
	
	// motor parameters
	g_motorTrqConst :ARRAY[1..4] OF LREAL :=[4(0.0292)];
	g_motorMaxCurrent :ARRAY[1..4] OF LREAL :=[4(1000)];//mA
	
	// motor and absEncoder direction
	g_motorDir :ARRAY[1..4] OF INT :=[1, 1, 1, -1];
	g_asbEncoderDir :ARRAY[1..4] OF INT :=[-1, 1, -1, -1];
																 
	// joint position limit
	g_minJntPos: ARRAY[1..4] OF LREAL:=[0,0*g_deg2Rad,0,0];
	g_maxJntPos: ARRAY[1..4] OF LREAL:=[0.37,32*g_deg2Rad,0.23,0.18];
		
	// joint motion velocity 
	g_jntCtrlMotionVel :ARRAY[1..7] OF LREAL :=[0.015,2*g_deg2Rad,0.01,0.0075];
	

END_VAR

// ---- GVLs/Configs/Robot3/GVL_ArmDynamics_3.TcGVL
{attribute 'global_init_slot' := '49992'}
{attribute 'qualified_only'}
// Robot3 Data
VAR_GLOBAL CONSTANT
	// arm gravity parameters
	(*graParam=[ 2.7244*m3 + 2.7244*m4 + 2.7244*m5 + 2.7244*m6 + 9.8*mx2 + 9.8*mx9,
				9.8*my2 + 9.8*my9,
				3.577*m4 + 3.577*m5 + 3.577*m6 + 0.49*m9 + 9.8*mx3 + 9.8*mx8
				1.5827*m4 + 1.5827*m5 + 1.5827*m6 + 9.8*my3 + 9.8*my8 + 9.8*mz4
				mz5-my4,	my5+mz6,  	mx4,   	mx5, 	mx6,   	my6
				preF2,   k2,   preF3,    k3,    preF5   k5]*)
	g_gravityParam :ARRAY[1..2, 1..16] OF REAL := 
		[ 6.2624762, -0.0007155225, 3.1411762, 0.48504608, -0.03459308, 0.025676297, 0.0000375, 0.0000351, -0.00001, -0.01593742,
		  7.7845001, 3195.0, 7.7845, 1902.6574, 2.5056201, 481.81768,
		  5.8820792, -0.0002385075, 2.9722568, 0.54387185, -0.037805167, 0.019637397, 0.000012500001, 0.0000117, -0.0000099999999, -0.013195626, 
		  10.732782, 2910.6441, 15.50438, 1786.0662, 2.1109713, 393.46033];
			
	// gravity deviation
	g_gravityDeviaion :ARRAY[1..2, 1..7] OF REAL :=
	[ 0.0, 0.0, 0.0, 0.0, 0.0, 0.0, 0.0, 
	 0.0, 0.0, 0.0, 0.0, 0.0, 0.0, 0.0];
	  
	// arm friction parameters [a1,b1,...a7,b7];
	// friction = a * gravity + b; only joint 5 and 6 is identified
	g_jntFrictionParam :ARRAY[1..2, 1..4] OF LREAL :=
	[ 0.18558566, 0.013430012, 0.1933446, 0.0056009337,
	  0.25838222, 0.0080955163, 0.3329508, 0.0062479093];
	g_maxJntFriction : Vec7d :=[0, 0, 0, 0, 0.05, 0.05, 0];
	
	//################ dynamic reference model parameters below ###########################
	// link mass [m1, m2, m3, m4, m5, m6, m7, m8, m9]
	g_linkMass :ARRAY[1..9] OF LREAL :=[2.676, 0.825, 0.547, 0.25, 0.195, 0.194, 0.05, 0.111, 0.09] ;
	
	// lin center of amss
	g_linkCOM :ARRAY[1..9,1..3] OF LREAL := [   1.376E-3,    -1.019E-3,  -81.464E-3,
										   90.622E-3,   -0.113E-3,  15.088E-3,
										   167.4E-3,    3.7E-3,     -0.438E-3,
										   0.1E-3,      98.49E-3,   -55.74E-3,
										   0.12E-3,     76.667E-3,  -36E-3,
										   0,           -61.63E-3,  27.3E-3,
										   0.06E-3,     -0.08E-3,   17.671E-3,
										   11E-3,       -3.364E-3,  39.265E-3,
										   143e-3,      0.495e-3,   24.253e-3];
	// link  inertial
    // [Ixx,Iyy,Izz, Ixy,Ixz, Iyz]
 	g_linkInertia :ARRAY[1..9,1..6] OF LREAL :=[  19.63E-3,   16.43E-3,  12.7E-3,   -0.3222E-3,    -0.667E-3,     -0.0268E-3,
												   1.017E-3,   6.637E-3,  5.935E-3,  -0.037E-3,     -0.238E-3,     0.06E-3,
												   0.161E-3,   9.572E-3,  9.586E-3,  0.0447E-3,     0.0277E-3,     0.465E-6,
												   0.992E-3,   0.707E-3,  0.335E-3,  0.2E-6,     2E-6,       0.224E-3,
												   0.402E-3,   0.25E-3,   0.186E-3,  0.002E-6,   -1.2E-6,    0.106E-3,
												   0.281E-3,   0.178E-3,  0.137E-3,  0.076E-6,   0.09E-6,    0.056E-3,
												   0.0255E-3,  0.0259E-3, 5.96E-6,0.34E-6,    -3E-9,      24E-9,
												   0.033E-3,   0.0976E-3, 0.126E-3,  3E-6,       -5E-6,      -0.162E-6,
												   4.9E-6,  0.757E-3,  0.760E-3,  2.6E-6,     -5.3E-6,    -18E-9];

	//################ DO NOT modify parameters below ###########################
	//  motor inertial at link size
	g_motorInertia :ARRAY[1..7] OF LREAL := [34.7E-7, 34.7E-7, 34.7E-7, 9.26E-7, 0.495E-7, 0.495E-7, 0.495E-7];
	
	// spring parameters
	// spring2 [L0, b1, b2, l1, r0]
	g_spring2Param :ARRAY[1..5] OF LREAL :=[101.6E-3, 14.5E-3, 15E-3, 172E-3, 31E-3];
	// spring3 [L0, b1, b2, l1, r0,d]
	g_spring3Param :ARRAY[1..6] OF LREAL :=[101.6E-3, 14E-3, 15E-3, 172E-3, 30E-3, 10E-3];
	// spring5 [L0, s1, L1, r0, beta]
	g_spring5Param :ARRAY[1..5] OF LREAL :=[34.93E-3, 34.3E-3, 100E-3, 12.5E-3, 32.02*g_deg2rad];
	
END_VAR

// ---- GVLs/Configs/Robot3/GVL_ArmJointCaliData_3.TcGVL
{attribute 'qualified_only'}
// Robot3 Data
VAR_GLOBAL CONSTANT									 
	// absolute encoder value at minimal joint positon
	g_minLinkEncoder :ARRAY[1..g_mArmNum, 1..g_mJntNum] OF DINT :=
		[5320292, 1637888, 16267012, 9121008, 16329376, 6965264, 0,
		 54048, 5138400, 12480240, 3380960, 9526944, 5270880, 0];
		 
	// absolute encoder value at maximum joint positon
	g_maxLinkEncoder :ARRAY[1..g_mArmNum, 1..g_mJntNum] OF DINT :=
		[16734116, 13586832, 3813732, 14235024, 11133568, 11256240, 0,
		 11534296, 16020072, 96940, 8157232, 13636784, 5270880, 0];
	
	// absolute encoder value at calibrated positon
	g_caliLinkEncoder :ARRAY[1..g_mArmNum, 1..g_mJntNum] OF DINT :=
		[2383568, 16504180, 1064304, 2073472, 6104944, 9016224, 13420592,
		 14507208, 2154776, 14028284, 15460608, 3197104, 7324448, 14964448];
	
	 // if absolute encoder value cross zeros within joint motion range
	 // NOTICE: joint 7 is always 0.
	g_linkEncZeroCross :ARRAY[1..g_mArmNum, 1..g_mJntNum] OF INT :=
		[1, 1, 1, 1, 1, 0, 1,
		 1, 1, 1, 1, 1, 0, 1];
		 
	// limit value of gripper hall sensor
	g_minHallSensorValue :ARRAY[1..2] OF DINT:=[2687067,3145824];
	g_maxHallSensorValue :ARRAY[1..2] OF DINT  :=[34800091,36635182];
		 
 	//################ DO NOT modify parameters below ###########################	
	// abolute encoder expanded limit buffer in case there is calibrtion error at limit position
	g_linkEncLimitBuffer : DINT := 100000;
	
	// flag if joint can rotate multiple cycles
	g_multipleCyclesJoint :ARRAY[1..g_mArmNum, 1..g_mJntNum] OF INT :=
		[0, 0, 0, 0, 0, 0, 1,
		 0, 0, 0, 0, 0, 0, 1];
		 
	// joint position at link encoder calibrated point
	g_linkEncCaliJntPos :ARRAY[1..g_mArmNum, 1..g_mJntNum] OF LREAL :=
		[0.0, -PI/2, 0.0, -pi, pi, -PI/2, 0.0,
		 0.0, -PI/2, 0.0, 0.0, pi, PI/2, 0.0];

END_VAR

// ---- GVLs/Configs/Robot3/GVL_CartJointCaliData_3.TcGVL
{attribute 'qualified_only'}
// Robot3 Data
VAR_GLOBAL CONSTANT
	(* cart joints are defiend in sequence as below
	[monitor lift, monitor rotate, armset, pedal] *)

	// absolute encoder value at minimal joint positon
	g_minLinkEncoder :ARRAY[1..4] OF DINT :=[10551943, 13637932, 8646306,11744290];
		 
	// absolute encoder value at maximum joint positon
	g_maxLinkEncoder :ARRAY[1..4] OF DINT :=[9057645, 16333724,7704162,10974938];
	
	// absolute encoder value at calibrated positon
	g_caliLinkEncoder :ARRAY[1..4] OF DINT :=[10551943, 13637932, 8646306,11744290];
	
	// if absolute encoder value cross zeros within joint motion range
	g_linkEncZeroCross :ARRAY[1..4] OF INT :=[0, 0, 0, 0];
		
	 //################ DO NOT modify parameters below ###########################
	// abolute encoder expanded limit buffer in case there is calibrtion error at limit position
	g_linkEncLimitBuffer : DINT := 100000;
	
	// flag if joint can rotate multiple cycles
	g_multipleCyclesJoint :ARRAY[1..4] OF INT :=[0, 0, 0, 0];
		 
	// joint position at link encoder calibrated point
	//TODO: joint2 calibration position need to be checked
	g_linkEncCaliJntPos :ARRAY[1..4] OF LREAL :=[0, 0*g_deg2Rad,0,0];

END_VAR

// ---- GVLs/Configs/Robot4/GVL_ArmDynamics_4.TcGVL
{attribute 'global_init_slot' := '49992'}
{attribute 'qualified_only'}
// Robot4 Data
VAR_GLOBAL CONSTANT
	// arm gravity parameters
	(*graParam=[ 2.7244*m3 + 2.7244*m4 + 2.7244*m5 + 2.7244*m6 + 9.8*mx2 + 9.8*mx9,
				9.8*my2 + 9.8*my9,
				3.577*m4 + 3.577*m5 + 3.577*m6 + 0.49*m9 + 9.8*mx3 + 9.8*mx8
				1.5827*m4 + 1.5827*m5 + 1.5827*m6 + 9.8*my3 + 9.8*my8 + 9.8*mz4
				mz5-my4,	my5+mz6,  	mx4,   	mx5, 	mx6,   	my6
				preF2,   k2,   preF3,    k3,    preF5   k5]*)
	g_gravityParam :ARRAY[1..2, 1..16] OF REAL := 
		[ 6.3392449, -0.0002385075, 3.0933659, 0.70940223, -0.034834554, 0.025682828, 0.0000375, 0.0000351, 0.00001, -0.015893351, 
		  7.7845, 3169.461, 15.57162, 1727.0133, 1.112, 542.07868,
		  6.2170758, -0.0002385075, 3.7070752, 0.91604839, -0.035060927, 0.025794159, 0.0000125, 0.0000117, -0.0000099999997, -0.015224975, 
		  9.9384443, 3075.5733, 15.14036, 2344.7901, 3.336, 467.18343];
			
	// gravity deviation
	g_gravityDeviaion :ARRAY[1..2, 1..7] OF REAL :=
	[ 0.0, 0.0, 0.0, 0.0, 0.0, 0.0, 0.0, 
	 0.0, 0.0, 0.0, 0.0, 0.0, 0.0, 0.0];
		  
	// arm friction parameters [a1,b1,...a7,b7];
	// friction = a * gravity + b; only joint 5 and 6 is identified
	g_jntFrictionParam :ARRAY[1..2, 1..4] OF LREAL :=
	[ 0.28041195, 0.0099822733, 0.34005097, 0.0093373104,
	0.25987842, 0.010223684, 0.24576829, 0.0051638863];
	g_maxJntFriction : Vec7d :=[0, 0, 0, 0, 0.05, 0.05, 0];
	
	//################ dynamic reference model parameters below ###########################
	// link mass [m1, m2, m3, m4, m5, m6, m7, m8, m9]
	g_linkMass :ARRAY[1..9] OF LREAL :=[2.676, 0.825, 0.547, 0.25, 0.195, 0.194, 0.05, 0.111, 0.09] ;
	
	// lin center of amss
	g_linkCOM :ARRAY[1..9,1..3] OF LREAL := [   1.376E-3,    -1.019E-3,  -81.464E-3,
										   90.622E-3,   -0.113E-3,  15.088E-3,
										   167.4E-3,    3.7E-3,     -0.438E-3,
										   0.1E-3,      98.49E-3,   -55.74E-3,
										   0.12E-3,     76.667E-3,  -36E-3,
										   0,           -61.63E-3,  27.3E-3,
										   0.06E-3,     -0.08E-3,   17.671E-3,
										   11E-3,       -3.364E-3,  39.265E-3,
										   143e-3,      0.495e-3,   24.253e-3];
	// link  inertial
    // [Ixx,Iyy,Izz, Ixy,Ixz, Iyz]
 	g_linkInertia :ARRAY[1..9,1..6] OF LREAL :=[  19.63E-3,   16.43E-3,  12.7E-3,   -0.3222E-3,    -0.667E-3,     -0.0268E-3,
												   1.017E-3,   6.637E-3,  5.935E-3,  -0.037E-3,     -0.238E-3,     0.06E-3,
												   0.161E-3,   9.572E-3,  9.586E-3,  0.0447E-3,     0.0277E-3,     0.465E-6,
												   0.992E-3,   0.707E-3,  0.335E-3,  0.2E-6,     2E-6,       0.224E-3,
												   0.402E-3,   0.25E-3,   0.186E-3,  0.002E-6,   -1.2E-6,    0.106E-3,
												   0.281E-3,   0.178E-3,  0.137E-3,  0.076E-6,   0.09E-6,    0.056E-3,
												   0.0255E-3,  0.0259E-3, 5.96E-6,0.34E-6,    -3E-9,      24E-9,
												   0.033E-3,   0.0976E-3, 0.126E-3,  3E-6,       -5E-6,      -0.162E-6,
												   4.9E-6,  0.757E-3,  0.760E-3,  2.6E-6,     -5.3E-6,    -18E-9];

	//################ DO NOT modify parameters below ###########################
	//  motor inertial at link size
	g_motorInertia :ARRAY[1..7] OF LREAL := [34.7E-7, 34.7E-7, 34.7E-7, 9.26E-7, 0.495E-7, 0.495E-7, 0.495E-7];
	
	// spring parameters
	// spring2 [L0, b1, b2, l1, r0]
	g_spring2Param :ARRAY[1..5] OF LREAL :=[101.6E-3, 14.5E-3, 15E-3, 172E-3, 31E-3];
	// spring3 [L0, b1, b2, l1, r0,d]
	g_spring3Param :ARRAY[1..6] OF LREAL :=[101.6E-3, 14E-3, 15E-3, 172E-3, 30E-3, 10E-3];
	// spring5 [L0, s1, L1, r0, beta]
	g_spring5Param :ARRAY[1..5] OF LREAL :=[34.93E-3, 34.3E-3, 100E-3, 12.5E-3, 32.02*g_deg2rad];
	
END_VAR

// ---- GVLs/Configs/Robot4/GVL_ArmJointCaliData_4.TcGVL
{attribute 'qualified_only'}
// Robot4 Data
VAR_GLOBAL CONSTANT										 
	// absolute encoder value at minimal joint positon
	g_minLinkEncoder :ARRAY[1..g_mArmNum, 1..g_mJntNum] OF DINT :=
		[14726704, 4156456, 15345668, 1991632, 16314208, 14415440, 0,
		 2048324, 9416252, 4526812, 8226032,651760 , 8965456, 0];
		 
	// absolute encoder value at maximum joint positon
	g_maxLinkEncoder :ARRAY[1..g_mArmNum, 1..g_mJntNum] OF DINT :=
		[8963928, 15089072, 1747256, 7226288, 12212368, 1891360, 16777216,
		 13022120, 3582816, 8511152, 13355760, 13305856, 13284352	, 16777216];
	
	// absolute encoder value at calibrated positon
	g_caliLinkEncoder :ARRAY[1..g_mArmNum, 1..g_mJntNum] OF DINT :=
		[11829704, 1302576, 105152, 11634960, 5974256, 16596400, 9523824,
		 15937604, 6523036, 10129420, 3988720, 7037424, 11098016, 8939696];
	
	 // if absolute encoder value cross zeros within joint motion range
	 // NOTICE: joint 7 is always 0.
	g_linkEncZeroCross :ARRAY[1..g_mArmNum, 1..g_mJntNum] OF INT :=
		[0, 1, 1, 1, 1, 1, 1,
		 1, 0, 0, 1, 0, 0, 1];
		 
	// limit value of gripper hall sensor
	g_minHallSensorValue :ARRAY[1..2] OF DINT:=[3211374,2687079];
	g_maxHallSensorValue :ARRAY[1..2] OF DINT  :=[44171868,48104169];
	 
	 //################ DO NOT modify parameters below ###########################	 
	// abolute encoder expanded limit buffer in case there is calibrtion error at limit position
	g_linkEncLimitBuffer : DINT := 100000;
	
	// flag if joint can rotate multiple cycles
	g_multipleCyclesJoint :ARRAY[1..g_mArmNum, 1..g_mJntNum] OF INT :=
		[0, 0, 0, 0, 0, 0, 1,
		 0, 0, 0, 0, 0, 0, 1];
		 
	// joint position at link encoder calibrated point
	g_linkEncCaliJntPos :ARRAY[1..g_mArmNum, 1..g_mJntNum] OF LREAL :=
		[0.0, -PI/2, 0.0, -pi, pi, -PI/2, 0.0,
		 0.0, -PI/2, 0.0, 0.0, pi, PI/2, 0.0];
		 
END_VAR

// ---- GVLs/Configs/Robot4/GVL_CartJointCaliData_4_1.TcGVL
{attribute 'qualified_only'}
// Robot4 Data
VAR_GLOBAL CONSTANT
	(* cart joints are defiend in sequence as below
	[monitor lift, monitor rotate, armset, pedal] *)
	
	// absolute encoder value at minimal joint positon
	g_minLinkEncoder :ARRAY[1..4] OF DINT :=[34123300, 5785968, 32214823,25465194];
		 
	// absolute encoder value at maximum joint positon
	g_maxLinkEncoder :ARRAY[1..4] OF DINT :=[32647732, 8246492,31272794,24686423];
	
	// absolute encoder value at calibrated positon
	g_caliLinkEncoder :ARRAY[1..4] OF DINT :=[34123300, 5785968, 32214823,25465194];
	
	// if absolute encoder value cross zeros within joint motion range
	g_linkEncZeroCross :ARRAY[1..4] OF INT :=[0, 0, 0, 0];
	
	//################ DO NOT modify parameters below ###########################
	// abolute encoder expanded limit buffer in case there is calibrtion error at limit position
	g_linkEncLimitBuffer : DINT := 100000;
	
	// flag if joint can rotate multiple cycles
	g_multipleCyclesJoint :ARRAY[1..4] OF INT :=[0, 0, 0, 0];
		 
	// joint position at link encoder calibrated point
	//TODO: joint2 calibration position need to be checked
	g_linkEncCaliJntPos :ARRAY[1..4] OF LREAL :=[0, 0*g_deg2Rad,0,0];

END_VAR

// ---- GVLs/Configs/Robot5/GVL_ArmDynamics_5.TcGVL
{attribute 'global_init_slot' := '49992'}
{attribute 'qualified_only'}
// Robot5 Data
VAR_GLOBAL CONSTANT
	// arm gravity parameters
	(*graParam=[ 2.7244*m3 + 2.7244*m4 + 2.7244*m5 + 2.7244*m6 + 9.8*mx2 + 9.8*mx9,
				9.8*my2 + 9.8*my9,
				3.577*m4 + 3.577*m5 + 3.577*m6 + 0.49*m9 + 9.8*mx3 + 9.8*mx8
				1.5827*m4 + 1.5827*m5 + 1.5827*m6 + 9.8*my3 + 9.8*my8 + 9.8*mz4
				mz5-my4,	my5+mz6,  	mx4,   	mx5, 	mx6,   	my6
				preF2,   k2,   preF3,    k3,    preF5   k5]*)
	g_gravityParam :ARRAY[1..2, 1..16] OF REAL := 
		[  6.233821, -0.0007155225, 2.1490133, 0.48504608, -0.04459068, 0.026744535, 0.0000125, 0.0000117, -0.00001, -0.016609005, 
		  7.7845, 3195.0, 7.7845, 1307.2023, 1.112, 559.81848,
		  6.1554212, -0.0007155225, 2.7407729, 0.48504608, -0.036823967, 0.023888653, 0.0000375, 0.0000117, -0.00001, -0.016609005, 
		  7.7845252, 3194.9998, 7.7845, 1621.7158, 3.336, 454.73229];
			
	// gravity deviation
	g_gravityDeviaion :ARRAY[1..2, 1..7] OF REAL :=
	[ 0.0, 0.0, 0.0, 0.0, 0.0, 0.0, 0.0, 
	 0.0, 0.0, 0.0, 0.0, 0.0, 0.0, 0.0];
	
	// arm friction parameters [a1,b1,...a7,b7];
	// friction = a * gravity + b; only joint 5 and 6 is identified
	g_jntFrictionParam :ARRAY[1..2, 1..4] OF LREAL :=
	[0.26783306, 0.010838125, 0.16823959, 0.014497874,
	 0.23963001, 0.010367281, 0.32339166, 0.0044046397];
	g_maxJntFriction : Vec7d :=[0, 0, 0, 0, 0.05, 0.05, 0];

	//################ dynamic reference model parameters below ###########################
	// link mass [m1, m2, m3, m4, m5, m6, m7, m8, m9]
	g_linkMass :ARRAY[1..9] OF LREAL :=[2.676, 0.825, 0.547, 0.25, 0.195, 0.194, 0.05, 0.111, 0.09] ;
	
	// lin center of amss
	g_linkCOM :ARRAY[1..9,1..3] OF LREAL := [   1.376E-3,    -1.019E-3,  -81.464E-3,
										   90.622E-3,   -0.113E-3,  15.088E-3,
										   167.4E-3,    3.7E-3,     -0.438E-3,
										   0.1E-3,      98.49E-3,   -55.74E-3,
										   0.12E-3,     76.667E-3,  -36E-3,
										   0,           -61.63E-3,  27.3E-3,
										   0.06E-3,     -0.08E-3,   17.671E-3,
										   11E-3,       -3.364E-3,  39.265E-3,
										   143e-3,      0.495e-3,   24.253e-3];
	// link  inertial
    // [Ixx,Iyy,Izz, Ixy,Ixz, Iyz]
 	g_linkInertia :ARRAY[1..9,1..6] OF LREAL :=[  19.63E-3,   16.43E-3,  12.7E-3,   -0.3222E-3,    -0.667E-3,     -0.0268E-3,
												   1.017E-3,   6.637E-3,  5.935E-3,  -0.037E-3,     -0.238E-3,     0.06E-3,
												   0.161E-3,   9.572E-3,  9.586E-3,  0.0447E-3,     0.0277E-3,     0.465E-6,
												   0.992E-3,   0.707E-3,  0.335E-3,  0.2E-6,     2E-6,       0.224E-3,
												   0.402E-3,   0.25E-3,   0.186E-3,  0.002E-6,   -1.2E-6,    0.106E-3,
												   0.281E-3,   0.178E-3,  0.137E-3,  0.076E-6,   0.09E-6,    0.056E-3,
												   0.0255E-3,  0.0259E-3, 5.96E-6,0.34E-6,    -3E-9,      24E-9,
												   0.033E-3,   0.0976E-3, 0.126E-3,  3E-6,       -5E-6,      -0.162E-6,
												   4.9E-6,  0.757E-3,  0.760E-3,  2.6E-6,     -5.3E-6,    -18E-9];

	//################ DO NOT modify parameters below ###########################
	//  motor inertial at link size
	g_motorInertia :ARRAY[1..7] OF LREAL := [34.7E-7, 34.7E-7, 34.7E-7, 9.26E-7, 0.495E-7, 0.495E-7, 0.495E-7];
	
	// spring parameters
	// spring2 [L0, b1, b2, l1, r0]
	g_spring2Param :ARRAY[1..5] OF LREAL :=[101.6E-3, 14.5E-3, 15E-3, 172E-3, 31E-3];
	// spring3 [L0, b1, b2, l1, r0,d]
	g_spring3Param :ARRAY[1..6] OF LREAL :=[101.6E-3, 14E-3, 15E-3, 172E-3, 30E-3, 10E-3];
	// spring5 [L0, s1, L1, r0, beta]
	g_spring5Param :ARRAY[1..5] OF LREAL :=[34.93E-3, 34.3E-3, 100E-3, 12.5E-3, 32.02*g_deg2rad];
	
END_VAR

// ---- GVLs/Configs/Robot5/GVL_ArmJointCaliData_5.TcGVL
{attribute 'qualified_only'}
// Robot5 Data
VAR_GLOBAL CONSTANT
	// absolute encoder value at minimal joint positon
	g_minLinkEncoder :ARRAY[1..g_mArmNum, 1..g_mJntNum] OF DINT :=
		[3330608, 6592612, 11754876, 8357648, 7032320, 3206208, 0,
		 14145556, 9942668, 4526812, 4839456,3252816 , 11705152, 0];
		 
	// absolute encoder value at maximum joint positon
	g_maxLinkEncoder :ARRAY[1..g_mArmNum, 1..g_mJntNum] OF DINT :=
		[9148752, 724532, 16056044, 13808640, 2987504, 7442528, 16777216,
		 3137384, 4088172, 8898876, 10199744, 15896032, 16050256, 16777216];
	
	// absolute encoder value at calibrated positon
	g_caliLinkEncoder :ARRAY[1..g_mArmNum, 1..g_mJntNum] OF DINT :=
		[6250820, 3647692, 13311308, 1419280, 13380032, 5208832, 11610128,
		 236924, 7059956, 5977404, 566400, 9673872, 13718496, 14927904];
	
	 // if absolute encoder value cross zeros within joint motion range
	 // NOTICE: joint 7 is always 0.
	g_linkEncZeroCross :ARRAY[1..g_mArmNum, 1..g_mJntNum] OF INT :=
		[0, 0, 0, 1, 1, 0, 1,
		 1, 0, 0, 1, 0, 0, 1];
		 
	// limit value of gripper hall sensor
	g_minHallSensorValue :ARRAY[1..2] OF DINT:=[3801219,2818152];
	g_maxHallSensorValue :ARRAY[1..2] OF DINT  :=[45023889,41878148];
	
	 //################ DO NOT modify parameters below ###########################
	// abolute encoder expanded limit buffer in case there is calibrtion error at limit position
	g_linkEncLimitBuffer : DINT := 100000;
	
	// flag if joint can rotate multiple cycles
	g_multipleCyclesJoint :ARRAY[1..g_mArmNum, 1..g_mJntNum] OF INT :=
		[0, 0, 0, 0, 0, 0, 1,
		 0, 0, 0, 0, 0, 0, 1];
		 
	// joint position at link encoder calibrated point
	g_linkEncCaliJntPos :ARRAY[1..g_mArmNum, 1..g_mJntNum] OF LREAL :=
		[0.0, -PI/2, 0.0, -pi, pi, -PI/2, 0.0,
		 0.0, -PI/2, 0.0, 0.0, pi, PI/2, 0.0];
		 
END_VAR

// ---- GVLs/Configs/Robot5/GVL_CartJointCaliData_5.TcGVL
{attribute 'qualified_only'}
// Robot5 Data
VAR_GLOBAL CONSTANT
	(* cart joints are defiend in sequence as below
	[monitor lift, monitor rotate, armset, pedal] *)
	
	// absolute encoder value at minimal joint positon
	g_minLinkEncoder :ARRAY[1..4] OF DINT :=[54146051, 12890812, 50227236,48935748];
		 
	// absolute encoder value at maximum joint positon
	g_maxLinkEncoder :ARRAY[1..4] OF DINT :=[52631155, 15542320,49285521,48159780];
	
	// absolute encoder value at calibrated positon
	g_caliLinkEncoder :ARRAY[1..4] OF DINT :=[54146051, 12890812, 50227236, 48935748];
	
	// if absolute encoder value cross zeros within joint motion range
	g_linkEncZeroCross :ARRAY[1..4] OF INT :=[0, 0, 0, 0];
	
	 //################ DO NOT modify parameters below ###########################
	// abolute encoder expanded limit buffer in case there is calibrtion error at limit position
	g_linkEncLimitBuffer : DINT := 100000;
	
	// flag if joint can rotate multiple cycles
	g_multipleCyclesJoint :ARRAY[1..4] OF INT :=[0, 0, 0, 0];
		 
	// joint position at link encoder calibrated point
	//TODO: joint2 calibration position need to be checked
	g_linkEncCaliJntPos :ARRAY[1..4] OF LREAL :=[0, 0*g_deg2Rad,0,0];

END_VAR

// ---- GVLs/Configs/Robot6/GVL_ArmDynamics_6.TcGVL
{attribute 'global_init_slot' := '49992'}
{attribute 'qualified_only'}
// Robot5 Data
VAR_GLOBAL CONSTANT
	// arm gravity parameters
	(*graParam=[ 2.7244*m3 + 2.7244*m4 + 2.7244*m5 + 2.7244*m6 + 9.8*mx2 + 9.8*mx9,
				9.8*my2 + 9.8*my9,
				3.577*m4 + 3.577*m5 + 3.577*m6 + 0.49*m9 + 9.8*mx3 + 9.8*mx8
				1.5827*m4 + 1.5827*m5 + 1.5827*m6 + 9.8*my3 + 9.8*my8 + 9.8*mz4
				mz5-my4,	my5+mz6,  	mx4,   	mx5, 	mx6,   	my6
				preF2,   k2,   preF3,    k3,    preF5   k5]*)
	g_gravityParam :ARRAY[1..2, 1..16] OF REAL := 
		[   5.7568045, -0.0007155225, 2.4474536, 0.48504608, -0.038756411, 0.023437688, 0.0000125, 0.0000117, 0.00001, -0.012844057, 
			12.442675, 2768.2548, 7.7845, 1404.7225, 1.1120001, 450.6766,
		  5.0678259, -0.0007155225, 3.4758647, 0.58104905, -0.038315725, 0.022496083, 0.0000125, 0.0000117, 0.00001, -0.013577169, 
			14.860859, 2540.3644, 14.374433, 1835.7932, 3.336, 377.86767];
			
	// gravity deviation
	g_gravityDeviaion :ARRAY[1..2, 1..7] OF REAL :=
	[ 0.0, 0.0, 0.0, 0.0, 0.0, 0.0, 0.0, 
	 0.0, 0.0, 0.0, 0.0, 0.0, 0.0, 0.0];
	 
	// arm friction parameters [a1,b1,...a7,b7];
	// friction = a * gravity + b; only joint 5 and 6 is identified
	g_jntFrictionParam :ARRAY[1..2, 1..4] OF LREAL :=
	[ 0.31293434, 0.0092686103, 0.40127329, 0.0065854475,
		0.27821857, 0.012357132, 0.34819478, 0.0068603075];
	g_maxJntFriction : Vec7d :=[0, 0, 0, 0, 0.05, 0.05, 0];

	//################ dynamic reference model parameters below ###########################
	// link mass [m1, m2, m3, m4, m5, m6, m7, m8, m9]
	g_linkMass :ARRAY[1..9] OF LREAL :=[2.676, 0.825, 0.547, 0.25, 0.195, 0.194, 0.05, 0.111, 0.09] ;
	
	// lin center of amss
	g_linkCOM :ARRAY[1..9,1..3] OF LREAL := [   1.376E-3,    -1.019E-3,  -81.464E-3,
										   90.622E-3,   -0.113E-3,  15.088E-3,
										   167.4E-3,    3.7E-3,     -0.438E-3,
										   0.1E-3,      98.49E-3,   -55.74E-3,
										   0.12E-3,     76.667E-3,  -36E-3,
										   0,           -61.63E-3,  27.3E-3,
										   0.06E-3,     -0.08E-3,   17.671E-3,
										   11E-3,       -3.364E-3,  39.265E-3,
										   143e-3,      0.495e-3,   24.253e-3];
	// link  inertial
    // [Ixx,Iyy,Izz, Ixy,Ixz, Iyz]
 	g_linkInertia :ARRAY[1..9,1..6] OF LREAL :=[  19.63E-3,   16.43E-3,  12.7E-3,   -0.3222E-3,    -0.667E-3,     -0.0268E-3,
												   1.017E-3,   6.637E-3,  5.935E-3,  -0.037E-3,     -0.238E-3,     0.06E-3,
												   0.161E-3,   9.572E-3,  9.586E-3,  0.0447E-3,     0.0277E-3,     0.465E-6,
												   0.992E-3,   0.707E-3,  0.335E-3,  0.2E-6,     2E-6,       0.224E-3,
												   0.402E-3,   0.25E-3,   0.186E-3,  0.002E-6,   -1.2E-6,    0.106E-3,
												   0.281E-3,   0.178E-3,  0.137E-3,  0.076E-6,   0.09E-6,    0.056E-3,
												   0.0255E-3,  0.0259E-3, 5.96E-6,0.34E-6,    -3E-9,      24E-9,
												   0.033E-3,   0.0976E-3, 0.126E-3,  3E-6,       -5E-6,      -0.162E-6,
												   4.9E-6,  0.757E-3,  0.760E-3,  2.6E-6,     -5.3E-6,    -18E-9];

	//################ DO NOT modify parameters below ###########################
	//  motor inertial at link size
	g_motorInertia :ARRAY[1..7] OF LREAL := [34.7E-7, 34.7E-7, 34.7E-7, 9.26E-7, 0.495E-7, 0.495E-7, 0.495E-7];
	
	// spring parameters
	// spring2 [L0, b1, b2, l1, r0]
	g_spring2Param :ARRAY[1..5] OF LREAL :=[101.6E-3, 14.5E-3, 15E-3, 172E-3, 31E-3];
	// spring3 [L0, b1, b2, l1, r0,d]
	g_spring3Param :ARRAY[1..6] OF LREAL :=[101.6E-3, 14E-3, 15E-3, 172E-3, 30E-3, 10E-3];
	// spring5 [L0, s1, L1, r0, beta]
	g_spring5Param :ARRAY[1..5] OF LREAL :=[34.93E-3, 34.3E-3, 100E-3, 12.5E-3, 32.02*g_deg2rad];
	
END_VAR

// ---- GVLs/Configs/Robot6/GVL_ArmJointCaliData_6.TcGVL
{attribute 'qualified_only'}
// Robot6 Data
VAR_GLOBAL CONSTANT
	// absolute encoder value at minimal joint positon
	g_minLinkEncoder :ARRAY[1..g_mArmNum, 1..g_mJntNum] OF DINT :=
		[1649902, 14712379, 5702891, 766260, 2495547, 7638782, 0,
		 1757269, 13672745, 13392538, 10388322,13843344 , 8623602, 0];
		 
	// absolute encoder value at maximum joint positon
	g_maxLinkEncoder :ARRAY[1..g_mArmNum, 1..g_mJntNum] OF DINT :=
		[7456788, 3764682, 1296904, 12166927, 15179687, 11834650, 16777216,
		 7525236, 2790868, 1025347, 4881083, 11405392, 12859838, 16777216];
	
	// absolute encoder value at calibrated positon
	g_caliLinkEncoder :ARRAY[1..g_mArmNum, 1..g_mJntNum] OF DINT :=
		[4557300, 797200, 2811950, 4880000, 8625800, 9872400, 11909200,
		 4703860, 16527150, 14997024, 782650, 5321280, 10937800, 9004224];
	
	 // if absolute encoder value cross zeros within joint motion range
	 // NOTICE: joint 7 is always 0.
	g_linkEncZeroCross :ARRAY[1..g_mArmNum, 1..g_mJntNum] OF INT :=
		[0, 1, 0, 0, 0, 0, 1,
		 0, 1, 1, 1, 1, 0, 1];
		 
	// limit value of gripper hall sensor
	g_minHallSensorValue :ARRAY[1..2] OF DINT:=[3801219,2818152];
	g_maxHallSensorValue :ARRAY[1..2] OF DINT  :=[45023889,41878148];
	
	 //################ DO NOT modify parameters below ###########################
	// abolute encoder expanded limit buffer in case there is calibrtion error at limit position
	g_linkEncLimitBuffer : DINT := 100000;
	
	// flag if joint can rotate multiple cycles
	g_multipleCyclesJoint :ARRAY[1..g_mArmNum, 1..g_mJntNum] OF INT :=
		[0, 0, 0, 0, 0, 0, 1,
		 0, 0, 0, 0, 0, 0, 1];
		 
	// joint position at link encoder calibrated point
	g_linkEncCaliJntPos :ARRAY[1..g_mArmNum, 1..g_mJntNum] OF LREAL :=
		[0.0, -PI/2, 0.0, -pi, pi, -PI/2, 0.0,
		 0.0, -PI/2, 0.0, 0.0, pi, PI/2, 0.0];
		 
END_VAR

// ---- GVLs/Configs/Robot6/GVL_CartJointCaliData_6.TcGVL
{attribute 'qualified_only'}
// Robot6 Data
VAR_GLOBAL CONSTANT
	(* cart joints are defiend in sequence as below
	[monitor lift, monitor rotate, armset, pedal] *)
	
	// absolute encoder value at minimal joint positon
	g_minLinkEncoder :ARRAY[1..4] OF DINT :=[8324215, 3073088, 9822199,5580000];
		 
	// absolute encoder value at maximum joint positon
	g_maxLinkEncoder :ARRAY[1..4] OF DINT :=[6650464, 15542320,8563889,6455968];
	
	// absolute encoder value at calibrated positon
	g_caliLinkEncoder :ARRAY[1..4] OF DINT :=[8324215, 3073088, 9822199, 5580000];
	
	// if absolute encoder value cross zeros within joint motion range
	g_linkEncZeroCross :ARRAY[1..4] OF INT :=[0, 0, 0, 0];
	
	 //################ DO NOT modify parameters below ###########################
	// abolute encoder expanded limit buffer in case there is calibrtion error at limit position
	g_linkEncLimitBuffer : DINT := 100000;
	
	// flag if joint can rotate multiple cycles
	g_multipleCyclesJoint :ARRAY[1..4] OF INT :=[0, 0, 0, 0];
		 
	// joint position at link encoder calibrated point
	//TODO: joint2 calibration position need to be checked
	g_linkEncCaliJntPos :ARRAY[1..4] OF LREAL :=[0, 0,0,0];

END_VAR

// ---- GVLs/GVL_interactUI.TcGVL
{attribute 'qualified_only'}
VAR_GLOBAL
	g_uiParaReload:BOOL:=TRUE;
	
	//true :login；false:logout
	g_userLogged : BOOL;
	
	//master slave scaling : 3:1 , 2:1 , 3:2
	g_masterSlaveScaling : UINT;

	//arm is disable : arm left 1  and  arm right 2
	g_armIsDisbale : UINT;	
	
	//arm assignment method : 1 auto  , 2 manual
	g_armAssignMethod : UINT;
	
	//master arm  mapping  slave arm
	g_armDistributionInfo : ST_arm_distribution;  
	
	//plc definite shutdown
	g_plcPowerOffEnable : BOOL;
	
	//cart in manual adjustment
	g_cartInMotion : BOOL;
	
	//ergonomic control enable 
	g_ergonomicCtrl : ST_ergonCtrlEnable; 
	g_ergonomicCtrlEnableLast : ST_ergonCtrlEnable;
	
	//ergonomic control data
	g_ergonomicCtrlData : ST_ergonomicCtrlData; 

	//ui send reset fault
	g_uiResetFault : UINT;	
	
	//plc send ergonomic current joint position to UI
	g_ergonomicCurData : ST_ergonomicCtrlData;
	
	//head in
	g_surgonHeadIn : BOOL;
	
	//finger clutch on off
	g_fingerClutchOnOff : BOOL;
	
	//error id 
	g_errIdType3 : UDINT;
	g_errIdType2 : UDINT;
	g_errIdType1 : UDINT;
	g_errIdType0 : UDINT;
	
	//master arms and cart self check finshed
	g_masterSelfCheckFinshed : BOOL; 
		
	//PLC version information
	g_plcVersion : STRING;

	//stop button ui  : 0 master stop 			
	g_masterStopButton : UINT:=1;
		
	g_digitalZoom : UINT;
	g_hapticZoom : BOOL;
	g_fineTurnning : REAL;
	
